KUKA KRL program: EPS_2_25748_MH05A_A_20260121065902.src

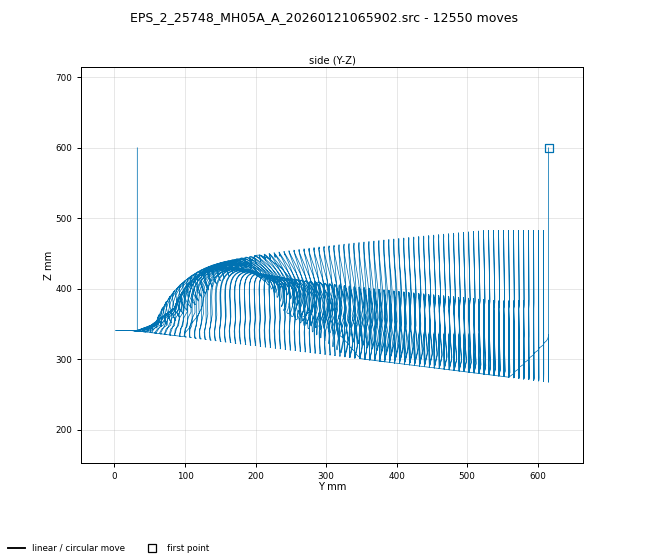
[picture p0: tool path of EPS_2_25748_MH05A_A_20260121065902.src, 12550 of 12552 moves have a stored position in this frame; points joined in program order, loops and branches not executed]
&ACCESS RVP
&REL 4
&COMMENT QRS 19112012
&PARAM EDITMASK = *
DEF PART()
EXT BAS (BAS_COMMAND :IN,REAL :IN )
INT I
BAS (#INITMOV,0 )

;KUKA QRS Post kuka4.cps  Date:22-06-2017 !

File_ID=3004

QRS_PRE_INIT()

;Init var - Until changes are made in qrs_pre_init
Outlet_Square_prg=0
Inlet_1_Square_prg=0
Inlet_2_Square_prg=0
Inlet_3_Square_prg=0
Inlet_4_Square_prg=0
Inlet_5_Square_prg=0

Outlet_1={X 0.000, Y 526.370, Z 382.500, B 0.000, E1 0.000 }
Inlet_1={X 0.000, Y 541.370, Z 332.500, B 0.000, E1 90.000 }
Inlet_2={X 0.000, Y 541.370, Z 332.500, B 0.000, E1 270.000 }
Outlet_1_type=201
Inlet_1_type=101
Inlet_2_type=101
;QRS#1=Sidecore dimensions
;QRS#2=200-8" PVC SDR 35
;QRS#3=100-4" PVC SDR 28
;QRS#4=100-4" PVC SDR 28
;QRS#5=
;QRS#6=
;QRS#7=
;QRS#8=
;QRS#9=12-08 PSX
;QRS#10=8QRS PSX
;QRS#11=8QRS PSX
;QRS#12=
;QRS#13=
;QRS#14=
;QRS#15=
;QRS#16=1220x127x762 2,5'
;QRS#17=EPS Height
;QRS#18=483
;QRS#19=*
;QRS#20= UPDATED VERSION 22-06-2017
;QRS#21=*
Outlet_Square=0100
Inlet_1_Square=045
Inlet_2_Square=045
Inlet_3_Square=0
Inlet_4_Square=0
Inlet_5_Square=0
Mill_Square=1
Outlet_Square_Prg=204
Inlet_1_Square_prg=201
Inlet_2_Square_prg=201

QRS_INIT()

$ADVANCE=5

; T1
PTP {E1 173.437,E2 173.437}
PTP {X 0,Y 615.487,A -85,B 0,C 180,E1 173.437,E2 173.437,E3 0,E4 0,E5 0,E6 0}
QRS_SPEED_INIT()
LIN {X 0,Y 615.487,Z 600,A -85,B 0,C 180,E1 173.437,E2 173.437,E3 0,E4 0,E5 0,E6 0} C_VEL
LIN {X 0,Y 615.487,Z 356.487,A -85,B 0,C 180,E1 173.437,E2 173.437} C_VEL
LIN {X 0,Y 615.487,Z 335.835,A -85,B 0,C 180,E1 173.437,E2 173.437} C_VEL
LIN {X 0,Y 615.487,Z 335.142,A -85,B 0,C 180,E1 173.425,E2 173.425} C_VEL
LIN {X 0,Y 615.489,Z 327.199,A -85,B 0,C 180,E1 173.165,E2 173.165} C_VEL
LIN {X 0,Y 615.468,Z 320.809,A -85,B 0,C 180,E1 170.802,E2 170.802} C_VEL
LIN {X 0,Y 615.487,Z 313.625,A -85,B 0,C 180,E1 168.14,E2 168.14} C_VEL
LIN {X 0,Y 615.472,Z 306.465,A -85,B 0,C 180,E1 165.452,E2 165.452} C_VEL
LIN {X 0,Y 615.459,Z 301.091,A -85,B 0,C 180,E1 163.414,E2 163.414} C_VEL
LIN {X 0,Y 615.449,Z 295.711,A -85,B 0,C 180,E1 161.354,E2 161.354} C_VEL
LIN {X 0,Y 615.488,Z 288.516,A -85,B 0,C 180,E1 158.569,E2 158.569} C_VEL
LIN {X 0,Y 615.439,Z 281.35,A -85,B 0,C 180,E1 155.727,E2 155.727} C_VEL
LIN {X 0,Y 615.424,Z 275.957,A -85,B 0,C 180,E1 153.554,E2 153.554} C_VEL
LIN {X 0,Y 615.496,Z 270.47,A -85,B 0,C 180,E1 151.344,E2 151.344} C_VEL
LIN {X 0,Y 615.454,Z 267.7,A -85,B 0,C 180,E1 150.211,E2 150.211} C_VEL
LIN {X 0,Y 615.419,Z 267.7,A -85,B 0,C 180,E1 147.54,E2 147.54} C_VEL
LIN {X 0,Y 615.453,Z 267.7,A -85,B 0,C 180,E1 145.184,E2 145.184} C_VEL
LIN {X 0,Y 615.487,Z 267.696,A -85,B 0,C 180,E1 142.759,E2 142.759} C_VEL
LIN {X 0,Y 615.437,Z 267.696,A -85,B 0,C 180,E1 140.248,E2 140.248} C_VEL
LIN {X 0,Y 615.459,Z 267.698,A -85,B 0,C 180,E1 137.646,E2 137.646} C_VEL
LIN {X 0,Y 615.492,Z 267.688,A -85,B 0,C 180,E1 134.934,E2 134.934} C_VEL
LIN {X 0,Y 615.453,Z 267.693,A -85,B 0,C 180,E1 132.356,E2 132.356} C_VEL
LIN {X 0,Y 615.497,Z 267.7,A -85,B 0,C 180,E1 129.75,E2 129.75} C_VEL
LIN {X 0,Y 615.478,Z 267.686,A -85,B 0,C 180,E1 126.938,E2 126.938} C_VEL
LIN {X 0,Y 615.495,Z 267.7,A -85,B 0,C 180,E1 124.022,E2 124.022} C_VEL
LIN {X 0,Y 615.484,Z 267.685,A -85,B 0,C 180,E1 121.088,E2 121.088} C_VEL
LIN {X 0,Y 615.494,Z 267.699,A -85,B 0,C 180,E1 118.454,E2 118.454} C_VEL
LIN {X 0,Y 615.485,Z 267.685,A -85,B 0,C 180,E1 115.571,E2 115.571} C_VEL
LIN {X 0,Y 615.492,Z 267.697,A -85,B 0,C 180,E1 112.844,E2 112.844} C_VEL
LIN {X 0,Y 615.476,Z 267.697,A -85,B 0,C 180,E1 110.558,E2 110.558} C_VEL
LIN {X 0,Y 615.468,Z 267.688,A -85,B 0,C 180,E1 107.958,E2 107.958} C_VEL
LIN {X 0,Y 615.497,Z 267.698,A -85,B 0,C 180,E1 105.226,E2 105.226} C_VEL
LIN {X 0,Y 615.447,Z 267.694,A -85,B 0,C 180,E1 102.531,E2 102.531} C_VEL
LIN {X 0,Y 615.489,Z 267.69,A -85,B 0,C 180,E1 99.862,E2 99.862} C_VEL
LIN {X 0,Y 615.455,Z 267.699,A -85,B 0,C 180,E1 97.216,E2 97.216} C_VEL
LIN {X 0,Y 615.445,Z 267.699,A -85,B 0,C 180,E1 95.242,E2 95.242} C_VEL
LIN {X 0,Y 615.436,Z 267.699,A -85,B 0,C 180,E1 93.273,E2 93.273} C_VEL
LIN {X 0,Y 615.428,Z 267.7,A -85,B 0,C 180,E1 91.309,E2 91.309} C_VEL
LIN {X 0,Y 615.426,Z 267.7,A -85,B 0,C 180,E1 89.346,E2 89.346} C_VEL
LIN {X 0,Y 615.429,Z 267.698,A -85,B 0,C 180,E1 87.382,E2 87.382} C_VEL
LIN {X 0,Y 615.433,Z 267.697,A -85,B 0,C 180,E1 85.415,E2 85.415} C_VEL
LIN {X 0,Y 615.436,Z 267.696,A -85,B 0,C 180,E1 83.443,E2 83.443} C_VEL
LIN {X 0,Y 615.465,Z 267.7,A -85,B 0,C 180,E1 80.801,E2 80.801} C_VEL
LIN {X 0,Y 615.481,Z 267.689,A -85,B 0,C 180,E1 78.139,E2 78.139} C_VEL
LIN {X 0,Y 615.455,Z 267.694,A -85,B 0,C 180,E1 75.45,E2 75.45} C_VEL
LIN {X 0,Y 615.489,Z 267.694,A -85,B 0,C 180,E1 72.729,E2 72.729} C_VEL
LIN {X 0,Y 615.467,Z 267.689,A -85,B 0,C 180,E1 69.966,E2 69.966} C_VEL
LIN {X 0,Y 615.474,Z 267.695,A -85,B 0,C 180,E1 67.653,E2 67.653} C_VEL
LIN {X 0,Y 615.483,Z 267.691,A -85,B 0,C 180,E1 65.008,E2 65.008} C_VEL
LIN {X 0,Y 615.484,Z 267.686,A -85,B 0,C 180,E1 62.823,E2 62.823} C_VEL
LIN {X 0,Y 615.481,Z 267.691,A -85,B 0,C 180,E1 60.204,E2 60.204} C_VEL
LIN {X 0,Y 615.476,Z 267.695,A -85,B 0,C 180,E1 57.542,E2 57.542} C_VEL
LIN {X 0,Y 615.471,Z 267.688,A -85,B 0,C 180,E1 55.184,E2 55.184} C_VEL
LIN {X 0,Y 615.495,Z 267.685,A -85,B 0,C 180,E1 52.758,E2 52.758} C_VEL
LIN {X 0,Y 615.464,Z 267.696,A -85,B 0,C 180,E1 49.912,E2 49.912} C_VEL
LIN {X 0,Y 615.451,Z 267.693,A -85,B 0,C 180,E1 47.644,E2 47.644} C_VEL
LIN {X 0,Y 615.493,Z 267.691,A -85,B 0,C 180,E1 44.932,E2 44.932} C_VEL
LIN {X 0,Y 615.456,Z 267.698,A -85,B 0,C 180,E1 42.354,E2 42.354} C_VEL
LIN {X 0,Y 615.435,Z 267.696,A -85,B 0,C 180,E1 39.753,E2 39.753} C_VEL
LIN {X 0,Y 615.487,Z 267.696,A -85,B 0,C 180,E1 37.241,E2 37.241} C_VEL
LIN {X 0,Y 615.437,Z 267.7,A -85,B 0,C 180,E1 34.693,E2 34.693} C_VEL
LIN {X 0,Y 615.418,Z 267.7,A -85,B 0,C 180,E1 32.32,E2 32.32} C_VEL
LIN {X 0,Y 615.467,Z 267.832,A -85,B 0,C 180,E1 29.693,E2 29.693} C_VEL
LIN {X 0,Y 615.464,Z 273.932,A -85,B 0,C 180,E1 27.177,E2 27.177} C_VEL
LIN {X 0,Y 615.444,Z 279.32,A -85,B 0,C 180,E1 24.992,E2 24.992} C_VEL
LIN {X 0,Y 615.435,Z 284.707,A -85,B 0,C 180,E1 22.845,E2 22.845} C_VEL
LIN {X 0,Y 615.435,Z 290.579,A -85,B 0,C 180,E1 20.543,E2 20.543} C_VEL
LIN {X 0,Y 615.494,Z 297.255,A -85,B 0,C 180,E1 17.956,E2 17.956} C_VEL
LIN {X 0,Y 615.458,Z 304.432,A -85,B 0,C 180,E1 15.226,E2 15.226} C_VEL
LIN {X 0,Y 615.458,Z 309.811,A -85,B 0,C 180,E1 13.201,E2 13.201} C_VEL
LIN {X 0,Y 615.486,Z 316.97,A -85,B 0,C 180,E1 10.526,E2 10.526} C_VEL
LIN {X 0,Y 615.488,Z 324.129,A -85,B 0,C 180,E1 7.875,E2 7.875} C_VEL
LIN {X 0,Y 615.484,Z 327.224,A -85,B 0,C 180,E1 6.736,E2 6.736} C_VEL
LIN {X 0,Y 615.489,Z 337.548,A -85,B 0,C 180,E1 6.391,E2 6.391} C_VEL
LIN {X 0,Y 615.493,Z 345.958,A -85,B 0,C 180,E1 5.98,E2 5.98} C_VEL
LIN {X 0,Y 615.473,Z 353.687,A -85,B 0,C 180,E1 5.487,E2 5.487} C_VEL
LIN {X 0,Y 615.479,Z 360.528,A -85,B 0,C 180,E1 4.912,E2 4.912} C_VEL
LIN {X 0,Y 615.497,Z 366.675,A -85,B 0,C 180,E1 4.255,E2 4.255} C_VEL
LIN {X 0,Y 615.497,Z 371.521,A -85,B 0,C 180,E1 3.6,E2 3.6} C_VEL
LIN {X 0,Y 615.496,Z 375.254,A -85,B 0,C 180,E1 2.944,E2 2.944} C_VEL
LIN {X 0,Y 615.5,Z 379.232,A -85,B 0,C 180,E1 1.962,E2 1.962} C_VEL
LIN {X 0,Y 615.495,Z 380.966,A -85,B 0,C 180,E1 1.308,E2 1.308} C_VEL
LIN {X 0,Y 615.496,Z 382.005,A -85,B 0,C 180,E1 0.653,E2 0.653} C_VEL
LIN {X 0,Y 615.495,Z 382.384,A -85,B 0,C 180,E1 -0.001,E2 -0.001} C_VEL
LIN {X 0,Y 615.496,Z 382.104,A -85,B 0,C 180,E1 -0.655,E2 -0.655} C_VEL
LIN {X 0,Y 615.497,Z 381.164,A -85,B 0,C 180,E1 -1.309,E2 -1.309} C_VEL
LIN {X 0,Y 615.5,Z 379.533,A -85,B 0,C 180,E1 -1.964,E2 -1.964} C_VEL
LIN {X 0,Y 615.498,Z 375.659,A -85,B 0,C 180,E1 -2.946,E2 -2.946} C_VEL
LIN {X 0,Y 615.5,Z 371.006,A -85,B 0,C 180,E1 -3.765,E2 -3.765} C_VEL
LIN {X 0,Y 615.498,Z 366.023,A -85,B 0,C 180,E1 -4.421,E2 -4.421} C_VEL
LIN {X 0,Y 615.481,Z 359.747,A -85,B 0,C 180,E1 -5.078,E2 -5.078} C_VEL
LIN {X 0,Y 615.481,Z 352.578,A -85,B 0,C 180,E1 -5.653,E2 -5.653} C_VEL
LIN {X 0,Y 615.485,Z 344.591,A -85,B 0,C 180,E1 -6.146,E2 -6.146} C_VEL
LIN {X 0,Y 615.487,Z 335.142,A -85,B 0,C 180,E1 -6.575,E2 -6.575} C_VEL
LIN {X 0,Y 615.489,Z 327.197,A -85,B 0,C 180,E1 -6.835,E2 -6.835} C_VEL
LIN {X 0,Y 615.468,Z 320.805,A -85,B 0,C 180,E1 -9.2,E2 -9.2} C_VEL
LIN {X 0,Y 615.487,Z 313.62,A -85,B 0,C 180,E1 -11.862,E2 -11.862} C_VEL
LIN {X 0,Y 615.471,Z 306.46,A -85,B 0,C 180,E1 -14.55,E2 -14.55} C_VEL
LIN {X 0,Y 615.459,Z 301.086,A -85,B 0,C 180,E1 -16.588,E2 -16.588} C_VEL
LIN {X 0,Y 615.449,Z 295.706,A -85,B 0,C 180,E1 -18.648,E2 -18.648} C_VEL
LIN {X 0,Y 615.488,Z 288.511,A -85,B 0,C 180,E1 -21.433,E2 -21.433} C_VEL
LIN {X 0,Y 615.439,Z 281.345,A -85,B 0,C 180,E1 -24.275,E2 -24.275} C_VEL
LIN {X 0,Y 615.424,Z 275.952,A -85,B 0,C 180,E1 -26.448,E2 -26.448} C_VEL
LIN {X 0,Y 615.494,Z 270.525,A -85,B 0,C 180,E1 -28.658,E2 -28.658} C_VEL
LIN {X 0,Y 615.474,Z 267.701,A -85,B 0,C 180,E1 -29.838,E2 -29.838} C_VEL
LIN {X 0,Y 615.483,Z 267.7,A -85,B 0,C 180,E1 -32.458,E2 -32.458} C_VEL
LIN {X 0,Y 615.499,Z 267.7,A -85,B 0,C 180,E1 -34.815,E2 -34.815} C_VEL
LIN {X 0,Y 615.494,Z 267.696,A -85,B 0,C 180,E1 -37.242,E2 -37.242} C_VEL
LIN {X 0,Y 615.497,Z 267.7,A -85,B 0,C 180,E1 -40.09,E2 -40.09} C_VEL
LIN {X 0,Y 615.492,Z 267.699,A -85,B 0,C 180,E1 -43.048,E2 -43.048} C_VEL
LIN {X 0,Y 615.474,Z 267.7,A -85,B 0,C 180,E1 -45.849,E2 -45.849} C_VEL
LIN {X 0,Y 615.495,Z 267.7,A -85,B 0,C 180,E1 -48.527,E2 -48.527} C_VEL
LIN {X 0,Y 615.489,Z 267.697,A -85,B 0,C 180,E1 -51.096,E2 -51.096} C_VEL
LIN {X 0,Y 615.49,Z 267.7,A -85,B 0,C 180,E1 -53.575,E2 -53.575} C_VEL
LIN {X 0,Y 615.484,Z 267.698,A -85,B 0,C 180,E1 -56.467,E2 -56.467} C_VEL
LIN {X 0,Y 615.487,Z 267.701,A -85,B 0,C 180,E1 -59.08,E2 -59.08} C_VEL
LIN {X 0,Y 615.475,Z 267.7,A -85,B 0,C 180,E1 -61.553,E2 -61.553} C_VEL
LIN {X 0,Y 615.499,Z 267.84,A -85,B 0,C 180,E1 -62.593,E2 -62.593} C_VEL
LIN {X 0,Y 615.489,Z 285.437,A -85,B 0,C 180,E1 -65.369,E2 -65.369} C_VEL
LIN {X 0,Y 615.479,Z 303.892,A -85,B 0,C 180,E1 -68.216,E2 -68.216} C_VEL
LIN {X 0,Y 615.48,Z 322.328,A -85,B 0,C 180,E1 -71.008,E2 -71.008} C_VEL
LIN {X 0,Y 615.475,Z 339.53,A -85,B 0,C 180,E1 -73.574,E2 -73.574} C_VEL
LIN {X 0,Y 615.493,Z 357.991,A -85,B 0,C 180,E1 -76.294,E2 -76.294} C_VEL
LIN {X 0,Y 615.497,Z 371.777,A -85,B 0,C 180,E1 -78.306,E2 -78.306} C_VEL
LIN {X 0,Y 615.48,Z 386.239,A -85,B 0,C 180,E1 -78.557,E2 -78.557} C_VEL
LIN {X 0,Y 615.474,Z 399.368,A -85,B 0,C 180,E1 -78.923,E2 -78.923} C_VEL
LIN {X 0,Y 615.487,Z 411.143,A -85,B 0,C 180,E1 -79.384,E2 -79.384} C_VEL
LIN {X 0,Y 615.486,Z 422.574,A -85,B 0,C 180,E1 -79.972,E2 -79.972} C_VEL
LIN {X 0,Y 615.499,Z 434.02,A -85,B 0,C 180,E1 -80.718,E2 -80.718} C_VEL
LIN {X 0,Y 615.498,Z 443.257,A -85,B 0,C 180,E1 -81.463,E2 -81.463} C_VEL
LIN {X 0,Y 615.5,Z 451.653,A -85,B 0,C 180,E1 -82.29,E2 -82.29} C_VEL
LIN {X 0,Y 615.497,Z 459.691,A -85,B 0,C 180,E1 -83.259,E2 -83.259} C_VEL
LIN {X 0,Y 615.499,Z 465.422,A -85,B 0,C 180,E1 -84.102,E2 -84.102} C_VEL
LIN {X 0,Y 615.496,Z 470.872,A -85,B 0,C 180,E1 -85.087,E2 -85.087} C_VEL
LIN {X 0,Y 615.497,Z 475.141,A -85,B 0,C 180,E1 -86.072,E2 -86.072} C_VEL
LIN {X 0,Y 615.494,Z 477.399,A -85,B 0,C 180,E1 -86.727,E2 -86.727} C_VEL
LIN {X 0,Y 615.497,Z 479.233,A -85,B 0,C 180,E1 -87.382,E2 -87.382} C_VEL
LIN {X 0,Y 615.5,Z 480.607,A -85,B 0,C 180,E1 -88.037,E2 -88.037} C_VEL
LIN {X 0,Y 615.496,Z 482.173,A -85,B 0,C 180,E1 -89.346,E2 -89.346} C_VEL
LIN {X 0,Y 615.494,Z 482.389,A -85,B 0,C 180,E1 -90,E2 -90} C_VEL
LIN {X 0,Y 615.495,Z 481.58,A -85,B 0,C 180,E1 -91.309,E2 -91.309} C_VEL
LIN {X 0,Y 615.5,Z 480.607,A -85,B 0,C 180,E1 -91.963,E2 -91.963} C_VEL
LIN {X 0,Y 615.497,Z 479.233,A -85,B 0,C 180,E1 -92.618,E2 -92.618} C_VEL
LIN {X 0,Y 615.496,Z 476.349,A -85,B 0,C 180,E1 -93.601,E2 -93.601} C_VEL
LIN {X 0,Y 615.498,Z 472.441,A -85,B 0,C 180,E1 -94.584,E2 -94.584} C_VEL
LIN {X 0,Y 615.499,Z 467.405,A -85,B 0,C 180,E1 -95.57,E2 -95.57} C_VEL
LIN {X 0,Y 615.497,Z 460.871,A -85,B 0,C 180,E1 -96.583,E2 -96.583} C_VEL
LIN {X 0,Y 615.497,Z 453.133,A -85,B 0,C 180,E1 -97.545,E2 -97.545} C_VEL
LIN {X 0,Y 615.498,Z 445.044,A -85,B 0,C 180,E1 -98.371,E2 -98.371} C_VEL
LIN {X 0,Y 615.499,Z 435.167,A -85,B 0,C 180,E1 -99.199,E2 -99.199} C_VEL
LIN {X 0,Y 615.49,Z 423.98,A -85,B 0,C 180,E1 -99.945,E2 -99.945} C_VEL
LIN {X 0,Y 615.487,Z 413.021,A -85,B 0,C 180,E1 -100.527,E2 -100.527} C_VEL
LIN {X 0,Y 615.475,Z 400.543,A -85,B 0,C 180,E1 -101.038,E2 -101.038} C_VEL
LIN {X 0,Y 615.478,Z 388.064,A -85,B 0,C 180,E1 -101.402,E2 -101.402} C_VEL
LIN {X 0,Y 615.495,Z 374.459,A -85,B 0,C 180,E1 -101.652,E2 -101.652} C_VEL
LIN {X 0,Y 615.497,Z 371.777,A -85,B 0,C 180,E1 -101.694,E2 -101.694} C_VEL
LIN {X 0,Y 615.474,Z 352.245,A -85,B 0,C 180,E1 -104.549,E2 -104.549} C_VEL
LIN {X 0,Y 615.494,Z 333.841,A -85,B 0,C 180,E1 -107.27,E2 -107.27} C_VEL
LIN {X 0,Y 615.486,Z 315.416,A -85,B 0,C 180,E1 -110.033,E2 -110.033} C_VEL
LIN {X 0,Y 615.492,Z 298.599,A -85,B 0,C 180,E1 -112.595,E2 -112.595} C_VEL
LIN {X 0,Y 615.496,Z 279.441,A -85,B 0,C 180,E1 -115.57,E2 -115.57} C_VEL
LIN {X 0,Y 615.498,Z 267.695,A -85,B 0,C 180,E1 -117.453,E2 -117.453} C_VEL
LIN {X 0,Y 615.487,Z 267.7,A -85,B 0,C 180,E1 -120.16,E2 -120.16} C_VEL
LIN {X 0,Y 615.477,Z 267.7,A -85,B 0,C 180,E1 -122.458,E2 -122.458} C_VEL
LIN {X 0,Y 615.479,Z 267.699,A -85,B 0,C 180,E1 -124.816,E2 -124.816} C_VEL
LIN {X 0,Y 615.498,Z 267.697,A -85,B 0,C 180,E1 -127.242,E2 -127.242} C_VEL
LIN {X 0,Y 615.474,Z 267.7,A -85,B 0,C 180,E1 -130.087,E2 -130.087} C_VEL
LIN {X 0,Y 615.473,Z 267.701,A -85,B 0,C 180,E1 -132.355,E2 -132.355} C_VEL
LIN {X 0,Y 615.491,Z 267.699,A -85,B 0,C 180,E1 -135.068,E2 -135.068} C_VEL
LIN {X 0,Y 615.483,Z 267.701,A -85,B 0,C 180,E1 -137.921,E2 -137.921} C_VEL
LIN {X 0,Y 615.494,Z 267.7,A -85,B 0,C 180,E1 -140.25,E2 -140.25} C_VEL
LIN {X 0,Y 615.493,Z 267.697,A -85,B 0,C 180,E1 -143.063,E2 -143.063} C_VEL
LIN {X 0,Y 615.487,Z 267.699,A -85,B 0,C 180,E1 -145.3,E2 -145.3} C_VEL
LIN {X 0,Y 615.494,Z 267.701,A -85,B 0,C 180,E1 -147.669,E2 -147.669} C_VEL
LIN {X 0,Y 615.491,Z 267.747,A -85,B 0,C 180,E1 -150.545,E2 -150.545} C_VEL
LIN {X 0,Y 615.49,Z 272.137,A -85,B 0,C 180,E1 -152.084,E2 -152.084} C_VEL
LIN {X 0,Y 615.444,Z 279.315,A -85,B 0,C 180,E1 -155.006,E2 -155.006} C_VEL
LIN {X 0,Y 615.435,Z 284.702,A -85,B 0,C 180,E1 -157.153,E2 -157.153} C_VEL
LIN {X 0,Y 615.435,Z 290.579,A -85,B 0,C 180,E1 -159.457,E2 -159.457} C_VEL
LIN {X 0,Y 615.494,Z 297.25,A -85,B 0,C 180,E1 -162.043,E2 -162.043} C_VEL
LIN {X 0,Y 615.458,Z 304.428,A -85,B 0,C 180,E1 -164.773,E2 -164.773} C_VEL
LIN {X 0,Y 615.458,Z 309.806,A -85,B 0,C 180,E1 -166.797,E2 -166.797} C_VEL
LIN {X 0,Y 615.486,Z 316.966,A -85,B 0,C 180,E1 -169.472,E2 -169.472} C_VEL
LIN {X 0,Y 615.488,Z 324.125,A -85,B 0,C 180,E1 -172.124,E2 -172.124} C_VEL
LIN {X 0,Y 615.484,Z 327.223,A -85,B 0,C 180,E1 -173.264,E2 -173.264} C_VEL
LIN {X 0,Y 615.489,Z 337.51,A -85,B 0,C 180,E1 -173.607,E2 -173.607} C_VEL
LIN {X 0,Y 615.493,Z 345.927,A -85,B 0,C 180,E1 -174.019,E2 -174.019} C_VEL
LIN {X 0,Y 615.473,Z 353.663,A -85,B 0,C 180,E1 -174.511,E2 -174.511} C_VEL
LIN {X 0,Y 615.479,Z 360.51,A -85,B 0,C 180,E1 -175.086,E2 -175.086} C_VEL
LIN {X 0,Y 615.497,Z 366.661,A -85,B 0,C 180,E1 -175.743,E2 -175.743} C_VEL
LIN {X 0,Y 615.497,Z 371.51,A -85,B 0,C 180,E1 -176.399,E2 -176.399} C_VEL
LIN {X 0,Y 615.496,Z 375.246,A -85,B 0,C 180,E1 -177.054,E2 -177.054} C_VEL
LIN {X 0,Y 615.5,Z 379.226,A -85,B 0,C 180,E1 -178.036,E2 -178.036} C_VEL
LIN {X 0,Y 615.495,Z 380.962,A -85,B 0,C 180,E1 -178.691,E2 -178.691} C_VEL
LIN {X 0,Y 615.496,Z 382.003,A -85,B 0,C 180,E1 -179.345,E2 -179.345} C_VEL
LIN {X 0,Y 615.495,Z 382.384,A -85,B 0,C 180,E1 -179.999,E2 -179.999} C_VEL
LIN {X 0,Y 615.496,Z 382.106,A -85,B 0,C 180,E1 -180.653,E2 -180.653} C_VEL
LIN {X 0,Y 615.497,Z 381.167,A -85,B 0,C 180,E1 -181.308,E2 -181.308} C_VEL
LIN {X 0,Y 615.5,Z 379.538,A -85,B 0,C 180,E1 -181.962,E2 -181.962} C_VEL
LIN {X 0,Y 615.497,Z 377.17,A -85,B 0,C 180,E1 -182.617,E2 -182.617} C_VEL
LIN {X 0,Y 615.498,Z 372.077,A -85,B 0,C 180,E1 -183.6,E2 -183.6} C_VEL
LIN {X 0,Y 615.499,Z 366.038,A -85,B 0,C 180,E1 -184.42,E2 -184.42} C_VEL
LIN {X 0,Y 615.482,Z 359.765,A -85,B 0,C 180,E1 -185.076,E2 -185.076} C_VEL
LIN {X 0,Y 615.481,Z 352.603,A -85,B 0,C 180,E1 -185.651,E2 -185.651} C_VEL
LIN {X 0,Y 615.485,Z 344.622,A -85,B 0,C 180,E1 -186.144,E2 -186.144} C_VEL
LIN {X 0,Y 615.487,Z 335.142,A -85,B 0,C 180,E1 -186.575,E2 -186.575} C_VEL
LIN {X 0,Y 615.134,Z 331.885,A -85,B 0,C 180,E1 -186.751,E2 -186.751} C_VEL
LIN {X 0,Y 614.287,Z 329.277,A -85,B 0,C 180,E1 -187,E2 -187} C_VEL
LIN {X 0,Y 612.54,Z 326.422,A -85,B 0,C 180,E1 -187.454,E2 -187.454} C_VEL
LIN {X 0,Y 610.632,Z 324.727,A -85,B 0,C 180,E1 -187.981,E2 -187.981} C_VEL
LIN {X 0,Y 608.713,Z 322.769,A -85,B 0,C 180,E1 -188.74,E2 -188.74} C_VEL
LIN {X 0,Y 608.404,Z 321.715,A -85,B 0,C 180,E1 -189.128,E2 -189.128} C_VEL
LIN {X 0,Y 608.405,Z 315.822,A -85,B 0,C 180,E1 -191.324,E2 -191.324} C_VEL
LIN {X 0,Y 608.43,Z 308.603,A -85,B 0,C 180,E1 -194.037,E2 -194.037} C_VEL
LIN {X 0,Y 608.397,Z 301.383,A -85,B 0,C 180,E1 -196.785,E2 -196.785} C_VEL
LIN {X 0,Y 608.443,Z 294.164,A -85,B 0,C 180,E1 -199.57,E2 -199.57} C_VEL
LIN {X 0,Y 608.393,Z 286.81,A -85,B 0,C 180,E1 -202.46,E2 -202.46} C_VEL
LIN {X 0,Y 608.417,Z 281.529,A -85,B 0,C 180,E1 -204.571,E2 -204.571} C_VEL
LIN {X 0,Y 608.46,Z 275.067,A -85,B 0,C 180,E1 -207.203,E2 -207.203} C_VEL
LIN {X 0,Y 608.439,Z 268.694,A -85,B 0,C 180,E1 -209.78,E2 -209.78} C_VEL
LIN {X 0,Y 608.405,Z 268.695,A -85,B 0,C 180,E1 -212.514,E2 -212.514} C_VEL
LIN {X 0,Y 608.418,Z 268.698,A -85,B 0,C 180,E1 -214.901,E2 -214.901} C_VEL
LIN {X 0,Y 608.431,Z 268.691,A -85,B 0,C 180,E1 -217.747,E2 -217.747} C_VEL
LIN {X 0,Y 608.426,Z 268.694,A -85,B 0,C 180,E1 -220.326,E2 -220.326} C_VEL
LIN {X 0,Y 608.462,Z 268.688,A -85,B 0,C 180,E1 -223.308,E2 -223.308} C_VEL
LIN {X 0,Y 608.447,Z 268.693,A -85,B 0,C 180,E1 -226.128,E2 -226.128} C_VEL
LIN {X 0,Y 608.459,Z 268.69,A -85,B 0,C 180,E1 -228.823,E2 -228.823} C_VEL
LIN {X 0,Y 608.459,Z 268.688,A -85,B 0,C 180,E1 -231.411,E2 -231.411} C_VEL
LIN {X 0,Y 608.471,Z 268.694,A -85,B 0,C 180,E1 -233.949,E2 -233.949} C_VEL
LIN {X 0,Y 608.466,Z 268.69,A -85,B 0,C 180,E1 -236.329,E2 -236.329} C_VEL
LIN {X 0,Y 608.47,Z 268.686,A -85,B 0,C 180,E1 -238.726,E2 -238.726} C_VEL
LIN {X 0,Y 608.473,Z 268.691,A -85,B 0,C 180,E1 -241.377,E2 -241.377} C_VEL
LIN {X 0,Y 608.443,Z 268.692,A -85,B 0,C 180,E1 -243.964,E2 -243.964} C_VEL
LIN {X 0,Y 608.452,Z 268.691,A -85,B 0,C 180,E1 -246.876,E2 -246.876} C_VEL
LIN {X 0,Y 608.46,Z 268.695,A -85,B 0,C 180,E1 -249.319,E2 -249.319} C_VEL
LIN {X 0,Y 608.432,Z 268.691,A -85,B 0,C 180,E1 -251.828,E2 -251.828} C_VEL
LIN {X 0,Y 608.474,Z 268.691,A -85,B 0,C 180,E1 -254.594,E2 -254.594} C_VEL
LIN {X 0,Y 608.448,Z 268.69,A -85,B 0,C 180,E1 -257.322,E2 -257.322} C_VEL
LIN {X 0,Y 608.45,Z 268.691,A -85,B 0,C 180,E1 -260.023,E2 -260.023} C_VEL
LIN {X 0,Y 608.426,Z 268.697,A -85,B 0,C 180,E1 -262.7,E2 -262.7} C_VEL
LIN {X 0,Y 608.431,Z 268.695,A -85,B 0,C 180,E1 -264.698,E2 -264.698} C_VEL
LIN {X 0,Y 608.423,Z 268.692,A -85,B 0,C 180,E1 -267.352,E2 -267.352} C_VEL
LIN {X 0,Y 608.465,Z 268.697,A -85,B 0,C 180,E1 -270,E2 -270} C_VEL
LIN {X 0,Y 608.424,Z 268.692,A -85,B 0,C 180,E1 -272.648,E2 -272.648} C_VEL
LIN {X 0,Y 608.433,Z 268.695,A -85,B 0,C 180,E1 -275.302,E2 -275.302} C_VEL
LIN {X 0,Y 608.468,Z 268.69,A -85,B 0,C 180,E1 -277.967,E2 -277.967} C_VEL
LIN {X 0,Y 608.427,Z 268.692,A -85,B 0,C 180,E1 -280.651,E2 -280.651} C_VEL
LIN {X 0,Y 608.469,Z 268.694,A -85,B 0,C 180,E1 -283.356,E2 -283.356} C_VEL
LIN {X 0,Y 608.443,Z 268.689,A -85,B 0,C 180,E1 -286.094,E2 -286.094} C_VEL
LIN {X 0,Y 608.448,Z 268.699,A -85,B 0,C 180,E1 -288.87,E2 -288.87} C_VEL
LIN {X 0,Y 608.466,Z 268.687,A -85,B 0,C 180,E1 -291.692,E2 -291.692} C_VEL
LIN {X 0,Y 608.446,Z 268.699,A -85,B 0,C 180,E1 -294.571,E2 -294.571} C_VEL
LIN {X 0,Y 608.475,Z 268.686,A -85,B 0,C 180,E1 -297.21,E2 -297.21} C_VEL
LIN {X 0,Y 608.465,Z 268.692,A -85,B 0,C 180,E1 -299.974,E2 -299.974} C_VEL
LIN {X 0,Y 608.452,Z 268.692,A -85,B 0,C 180,E1 -302.523,E2 -302.523} C_VEL
LIN {X 0,Y 608.464,Z 268.687,A -85,B 0,C 180,E1 -304.91,E2 -304.91} C_VEL
LIN {X 0,Y 608.465,Z 268.696,A -85,B 0,C 180,E1 -307.747,E2 -307.747} C_VEL
LIN {X 0,Y 608.428,Z 268.693,A -85,B 0,C 180,E1 -310.328,E2 -310.328} C_VEL
LIN {X 0,Y 608.45,Z 268.691,A -85,B 0,C 180,E1 -312.96,E2 -312.96} C_VEL
LIN {X 0,Y 608.428,Z 268.695,A -85,B 0,C 180,E1 -315.739,E2 -315.739} C_VEL
LIN {X 0,Y 608.423,Z 268.693,A -85,B 0,C 180,E1 -317.937,E2 -317.937} C_VEL
LIN {X 0,Y 608.439,Z 268.694,A -85,B 0,C 180,E1 -320.706,E2 -320.706} C_VEL
LIN {X 0,Y 608.449,Z 268.696,A -85,B 0,C 180,E1 -323.086,E2 -323.086} C_VEL
LIN {X 0,Y 608.42,Z 268.693,A -85,B 0,C 180,E1 -325.529,E2 -325.529} C_VEL
LIN {X 0,Y 608.416,Z 268.693,A -85,B 0,C 180,E1 -327.904,E2 -327.904} C_VEL
LIN {X 0,Y 608.458,Z 268.865,A -85,B 0,C 180,E1 -330.317,E2 -330.317} C_VEL
LIN {X 0,Y 608.457,Z 274.849,A -85,B 0,C 180,E1 -332.797,E2 -332.797} C_VEL
LIN {X 0,Y 608.411,Z 281.306,A -85,B 0,C 180,E1 -335.428,E2 -335.428} C_VEL
LIN {X 0,Y 608.431,Z 288.521,A -85,B 0,C 180,E1 -338.308,E2 -338.308} C_VEL
LIN {X 0,Y 608.409,Z 295.737,A -85,B 0,C 180,E1 -341.13,E2 -341.13} C_VEL
LIN {X 0,Y 608.44,Z 302.953,A -85,B 0,C 180,E1 -343.907,E2 -343.907} C_VEL
LIN {X 0,Y 608.411,Z 310.169,A -85,B 0,C 180,E1 -346.643,E2 -346.643} C_VEL
LIN {X 0,Y 608.419,Z 317.385,A -85,B 0,C 180,E1 -349.35,E2 -349.35} C_VEL
LIN {X 0,Y 608.419,Z 324.602,A -85,B 0,C 180,E1 -352.033,E2 -352.033} C_VEL
LIN {X 0,Y 608.446,Z 327.892,A -85,B 0,C 180,E1 -353.187,E2 -353.187} C_VEL
LIN {X 0,Y 608.477,Z 338.104,A -85,B 0,C 180,E1 -353.535,E2 -353.535} C_VEL
LIN {X 0,Y 608.464,Z 346.487,A -85,B 0,C 180,E1 -353.951,E2 -353.951} C_VEL
LIN {X 0,Y 608.438,Z 355.268,A -85,B 0,C 180,E1 -354.533,E2 -354.533} C_VEL
LIN {X 0,Y 608.456,Z 362.738,A -85,B 0,C 180,E1 -355.197,E2 -355.197} C_VEL
LIN {X 0,Y 608.437,Z 368.565,A -85,B 0,C 180,E1 -355.861,E2 -355.861} C_VEL
LIN {X 0,Y 608.451,Z 372.073,A -85,B 0,C 180,E1 -356.359,E2 -356.359} C_VEL
LIN {X 0,Y 608.451,Z 375.824,A -85,B 0,C 180,E1 -357.021,E2 -357.021} C_VEL
LIN {X 0,Y 608.445,Z 379.829,A -85,B 0,C 180,E1 -358.015,E2 -358.015} C_VEL
LIN {X 0,Y 608.448,Z 381.57,A -85,B 0,C 180,E1 -358.677,E2 -358.677} C_VEL
LIN {X 0,Y 608.439,Z 382.615,A -85,B 0,C 180,E1 -359.339,E2 -359.339} C_VEL
LIN {X 0,Y 608.435,Z 382.995,A -85,B 0,C 180,E1 -360.001,E2 -360.001} C_VEL
LIN {X 0,Y 608.438,Z 382.713,A -85,B 0,C 180,E1 -360.663,E2 -360.663} C_VEL
LIN {X 0,Y 608.449,Z 381.766,A -85,B 0,C 180,E1 -361.325,E2 -361.325} C_VEL
LIN {X 0,Y 608.445,Z 380.126,A -85,B 0,C 180,E1 -361.987,E2 -361.987} C_VEL
LIN {X 0,Y 608.429,Z 377.742,A -85,B 0,C 180,E1 -362.649,E2 -362.649} C_VEL
LIN {X 0,Y 608.452,Z 372.614,A -85,B 0,C 180,E1 -363.643,E2 -363.643} C_VEL
LIN {X 0,Y 608.451,Z 366.548,A -85,B 0,C 180,E1 -364.473,E2 -364.473} C_VEL
LIN {X 0,Y 608.429,Z 360.244,A -85,B 0,C 180,E1 -365.137,E2 -365.137} C_VEL
LIN {X 0,Y 608.463,Z 353.082,A -85,B 0,C 180,E1 -365.718,E2 -365.718} C_VEL
LIN {X 0,Y 608.445,Z 345.091,A -85,B 0,C 180,E1 -366.217,E2 -366.217} C_VEL
LIN {X 0,Y 608.466,Z 336.237,A -85,B 0,C 180,E1 -366.633,E2 -366.633} C_VEL
LIN {X 0,Y 608.428,Z 327.701,A -85,B 0,C 180,E1 -366.91,E2 -366.91} C_VEL
LIN {X 0,Y 608.402,Z 321.231,A -85,B 0,C 180,E1 -369.308,E2 -369.308} C_VEL
LIN {X 0,Y 608.432,Z 314.012,A -85,B 0,C 180,E1 -372.001,E2 -372.001} C_VEL
LIN {X 0,Y 608.429,Z 306.793,A -85,B 0,C 180,E1 -374.722,E2 -374.722} C_VEL
LIN {X 0,Y 608.423,Z 299.574,A -85,B 0,C 180,E1 -377.478,E2 -377.478} C_VEL
LIN {X 0,Y 608.422,Z 292.354,A -85,B 0,C 180,E1 -380.276,E2 -380.276} C_VEL
LIN {X 0,Y 608.427,Z 285.134,A -85,B 0,C 180,E1 -383.126,E2 -383.126} C_VEL
LIN {X 0,Y 608.419,Z 277.914,A -85,B 0,C 180,E1 -386.037,E2 -386.037} C_VEL
LIN {X 0,Y 608.482,Z 271.589,A -85,B 0,C 180,E1 -388.621,E2 -388.621} C_VEL
LIN {X 0,Y 608.455,Z 268.696,A -85,B 0,C 180,E1 -389.841,E2 -389.841} C_VEL
LIN {X 0,Y 608.46,Z 268.696,A -85,B 0,C 180,E1 -392.522,E2 -392.522} C_VEL
LIN {X 0,Y 608.45,Z 268.696,A -85,B 0,C 180,E1 -395.278,E2 -395.278} C_VEL
LIN {X 0,Y 608.472,Z 268.694,A -85,B 0,C 180,E1 -397.747,E2 -397.747} C_VEL
LIN {X 0,Y 608.451,Z 268.696,A -85,B 0,C 180,E1 -400.329,E2 -400.329} C_VEL
LIN {X 0,Y 608.457,Z 268.696,A -85,B 0,C 180,E1 -402.96,E2 -402.96} C_VEL
LIN {X 0,Y 608.448,Z 268.696,A -85,B 0,C 180,E1 -405.738,E2 -405.738} C_VEL
LIN {X 0,Y 608.47,Z 268.694,A -85,B 0,C 180,E1 -408.658,E2 -408.658} C_VEL
LIN {X 0,Y 608.464,Z 268.696,A -85,B 0,C 180,E1 -411.761,E2 -411.761} C_VEL
LIN {X 0,Y 608.447,Z 268.697,A -85,B 0,C 180,E1 -413.955,E2 -413.955} C_VEL
LIN {X 0,Y 608.452,Z 268.695,A -85,B 0,C 180,E1 -416.328,E2 -416.328} C_VEL
LIN {X 0,Y 608.452,Z 268.696,A -85,B 0,C 180,E1 -418.732,E2 -418.732} C_VEL
LIN {X 0,Y 608.467,Z 268.694,A -85,B 0,C 180,E1 -421.382,E2 -421.382} C_VEL
LIN {X 0,Y 608.481,Z 268.705,A -85,B 0,C 180,E1 -422.39,E2 -422.39} C_VEL
LIN {X 0,Y 608.603,Z 280.287,A -85,B 0,C 180,E1 -424.254,E2 -424.254} C_VEL
LIN {X 0,Y 608.557,Z 298.245,A -85,B 0,C 180,E1 -427.078,E2 -427.078} C_VEL
LIN {X 0,Y 608.533,Z 316.593,A -85,B 0,C 180,E1 -429.904,E2 -429.904} C_VEL
LIN {X 0,Y 608.507,Z 335.055,A -85,B 0,C 180,E1 -432.698,E2 -432.698} C_VEL
LIN {X 0,Y 608.463,Z 353.518,A -85,B 0,C 180,E1 -435.45,E2 -435.45} C_VEL
LIN {X 0,Y 608.482,Z 371.981,A -85,B 0,C 180,E1 -438.17,E2 -438.17} C_VEL
LIN {X 0,Y 608.544,Z 387.264,A -85,B 0,C 180,E1 -438.445,E2 -438.445} C_VEL
LIN {X 0,Y 608.519,Z 399.925,A -85,B 0,C 180,E1 -438.809,E2 -438.809} C_VEL
LIN {X 0,Y 608.51,Z 411.635,A -85,B 0,C 180,E1 -439.277,E2 -439.277} C_VEL
LIN {X 0,Y 608.494,Z 422.755,A -85,B 0,C 180,E1 -439.855,E2 -439.855} C_VEL
LIN {X 0,Y 608.504,Z 434.251,A -85,B 0,C 180,E1 -440.611,E2 -440.611} C_VEL
LIN {X 0,Y 608.472,Z 443.536,A -85,B 0,C 180,E1 -441.364,E2 -441.364} C_VEL
LIN {X 0,Y 608.456,Z 451.989,A -85,B 0,C 180,E1 -442.2,E2 -442.2} C_VEL
LIN {X 0,Y 608.462,Z 460.235,A -85,B 0,C 180,E1 -443.201,E2 -443.201} C_VEL
LIN {X 0,Y 608.438,Z 466.876,A -85,B 0,C 180,E1 -444.199,E2 -444.199} C_VEL
LIN {X 0,Y 608.432,Z 472.95,A -85,B 0,C 180,E1 -445.362,E2 -445.362} C_VEL
LIN {X 0,Y 608.449,Z 476.896,A -85,B 0,C 180,E1 -446.358,E2 -446.358} C_VEL
LIN {X 0,Y 608.425,Z 479.809,A -85,B 0,C 180,E1 -447.352,E2 -447.352} C_VEL
LIN {X 0,Y 608.445,Z 481.201,A -85,B 0,C 180,E1 -448.014,E2 -448.014} C_VEL
LIN {X 0,Y 608.438,Z 482.783,A -85,B 0,C 180,E1 -449.338,E2 -449.338} C_VEL
LIN {X 0,Y 608.434,Z 483,A -85,B 0,C 180,E1 -450,E2 -450} C_VEL
LIN {X 0,Y 608.448,Z 482.184,A -85,B 0,C 180,E1 -451.324,E2 -451.324} C_VEL
LIN {X 0,Y 608.445,Z 481.201,A -85,B 0,C 180,E1 -451.986,E2 -451.986} C_VEL
LIN {X 0,Y 608.425,Z 479.809,A -85,B 0,C 180,E1 -452.648,E2 -452.648} C_VEL
LIN {X 0,Y 608.449,Z 476.896,A -85,B 0,C 180,E1 -453.642,E2 -453.642} C_VEL
LIN {X 0,Y 608.432,Z 472.95,A -85,B 0,C 180,E1 -454.638,E2 -454.638} C_VEL
LIN {X 0,Y 608.438,Z 466.876,A -85,B 0,C 180,E1 -455.801,E2 -455.801} C_VEL
LIN {X 0,Y 608.462,Z 460.235,A -85,B 0,C 180,E1 -456.799,E2 -456.799} C_VEL
LIN {X 0,Y 608.456,Z 451.989,A -85,B 0,C 180,E1 -457.8,E2 -457.8} C_VEL
LIN {X 0,Y 608.472,Z 443.536,A -85,B 0,C 180,E1 -458.636,E2 -458.636} C_VEL
LIN {X 0,Y 608.481,Z 433.09,A -85,B 0,C 180,E1 -459.473,E2 -459.473} C_VEL
LIN {X 0,Y 608.494,Z 422.754,A -85,B 0,C 180,E1 -460.145,E2 -460.145} C_VEL
LIN {X 0,Y 608.51,Z 411.635,A -85,B 0,C 180,E1 -460.723,E2 -460.723} C_VEL
LIN {X 0,Y 608.519,Z 399.926,A -85,B 0,C 180,E1 -461.191,E2 -461.191} C_VEL
LIN {X 0,Y 608.544,Z 387.265,A -85,B 0,C 180,E1 -461.555,E2 -461.555} C_VEL
LIN {X 0,Y 608.57,Z 374.597,A -85,B 0,C 180,E1 -461.786,E2 -461.786} C_VEL
LIN {X 0,Y 608.484,Z 371.981,A -85,B 0,C 180,E1 -461.83,E2 -461.83} C_VEL
LIN {X 0,Y 608.479,Z 352.364,A -85,B 0,C 180,E1 -464.72,E2 -464.72} C_VEL
LIN {X 0,Y 608.51,Z 333.901,A -85,B 0,C 180,E1 -467.475,E2 -467.475} C_VEL
LIN {X 0,Y 608.517,Z 315.439,A -85,B 0,C 180,E1 -470.272,E2 -470.272} C_VEL
LIN {X 0,Y 608.57,Z 298.131,A -85,B 0,C 180,E1 -472.939,E2 -472.939} C_VEL
LIN {X 0,Y 608.613,Z 280.271,A -85,B 0,C 180,E1 -475.748,E2 -475.748} C_VEL
LIN {X 0,Y 608.481,Z 268.705,A -85,B 0,C 180,E1 -477.61,E2 -477.61} C_VEL
LIN {X 0,Y 608.471,Z 268.693,A -85,B 0,C 180,E1 -480.545,E2 -480.545} C_VEL
LIN {X 0,Y 608.456,Z 268.695,A -85,B 0,C 180,E1 -482.88,E2 -482.88} C_VEL
LIN {X 0,Y 608.437,Z 268.7,A -85,B 0,C 180,E1 -485.278,E2 -485.278} C_VEL
LIN {X 0,Y 608.464,Z 268.694,A -85,B 0,C 180,E1 -487.747,E2 -487.747} C_VEL
LIN {X 0,Y 608.445,Z 268.697,A -85,B 0,C 180,E1 -490.328,E2 -490.328} C_VEL
LIN {X 0,Y 608.477,Z 268.692,A -85,B 0,C 180,E1 -493.309,E2 -493.309} C_VEL
LIN {X 0,Y 608.473,Z 268.694,A -85,B 0,C 180,E1 -496.13,E2 -496.13} C_VEL
LIN {X 0,Y 608.456,Z 268.695,A -85,B 0,C 180,E1 -498.823,E2 -498.823} C_VEL
LIN {X 0,Y 608.44,Z 268.698,A -85,B 0,C 180,E1 -501.409,E2 -501.409} C_VEL
LIN {X 0,Y 608.448,Z 268.696,A -85,B 0,C 180,E1 -503.955,E2 -503.955} C_VEL
LIN {X 0,Y 608.449,Z 268.697,A -85,B 0,C 180,E1 -506.328,E2 -506.328} C_VEL
LIN {X 0,Y 608.449,Z 268.699,A -85,B 0,C 180,E1 -508.733,E2 -508.733} C_VEL
LIN {X 0,Y 608.439,Z 268.809,A -85,B 0,C 180,E1 -510.646,E2 -510.646} C_VEL
LIN {X 0,Y 608.438,Z 274.857,A -85,B 0,C 180,E1 -512.801,E2 -512.801} C_VEL
LIN {X 0,Y 608.383,Z 281.301,A -85,B 0,C 180,E1 -515.425,E2 -515.425} C_VEL
LIN {X 0,Y 608.388,Z 286.713,A -85,B 0,C 180,E1 -517.591,E2 -517.591} C_VEL
LIN {X 0,Y 608.439,Z 293.928,A -85,B 0,C 180,E1 -520.428,E2 -520.428} C_VEL
LIN {X 0,Y 608.421,Z 299.34,A -85,B 0,C 180,E1 -522.522,E2 -522.522} C_VEL
LIN {X 0,Y 608.403,Z 304.752,A -85,B 0,C 180,E1 -524.592,E2 -524.592} C_VEL
LIN {X 0,Y 608.411,Z 310.164,A -85,B 0,C 180,E1 -526.642,E2 -526.642} C_VEL
LIN {X 0,Y 608.419,Z 317.38,A -85,B 0,C 180,E1 -529.349,E2 -529.349} C_VEL
LIN {X 0,Y 608.42,Z 324.597,A -85,B 0,C 180,E1 -532.032,E2 -532.032} C_VEL
LIN {X 0,Y 608.43,Z 327.839,A -85,B 0,C 180,E1 -533.186,E2 -533.186} C_VEL
LIN {X 0,Y 608.479,Z 338.067,A -85,B 0,C 180,E1 -533.533,E2 -533.533} C_VEL
LIN {X 0,Y 608.464,Z 346.462,A -85,B 0,C 180,E1 -533.949,E2 -533.949} C_VEL
LIN {X 0,Y 608.438,Z 355.246,A -85,B 0,C 180,E1 -534.531,E2 -534.531} C_VEL
LIN {X 0,Y 608.456,Z 362.72,A -85,B 0,C 180,E1 -535.196,E2 -535.196} C_VEL
LIN {X 0,Y 608.437,Z 368.553,A -85,B 0,C 180,E1 -535.859,E2 -535.859} C_VEL
LIN {X 0,Y 608.451,Z 372.062,A -85,B 0,C 180,E1 -536.357,E2 -536.357} C_VEL
LIN {X 0,Y 608.451,Z 375.815,A -85,B 0,C 180,E1 -537.02,E2 -537.02} C_VEL
LIN {X 0,Y 608.445,Z 379.822,A -85,B 0,C 180,E1 -538.013,E2 -538.013} C_VEL
LIN {X 0,Y 608.448,Z 381.566,A -85,B 0,C 180,E1 -538.675,E2 -538.675} C_VEL
LIN {X 0,Y 608.439,Z 382.614,A -85,B 0,C 180,E1 -539.337,E2 -539.337} C_VEL
LIN {X 0,Y 608.435,Z 382.995,A -85,B 0,C 180,E1 -539.999,E2 -539.999} C_VEL
LIN {X 0,Y 608.438,Z 382.715,A -85,B 0,C 180,E1 -540.661,E2 -540.661} C_VEL
LIN {X 0,Y 608.449,Z 381.77,A -85,B 0,C 180,E1 -541.323,E2 -541.323} C_VEL
LIN {X 0,Y 608.445,Z 380.131,A -85,B 0,C 180,E1 -541.985,E2 -541.985} C_VEL
LIN {X 0,Y 608.429,Z 377.749,A -85,B 0,C 180,E1 -542.647,E2 -542.647} C_VEL
LIN {X 0,Y 608.452,Z 372.624,A -85,B 0,C 180,E1 -543.641,E2 -543.641} C_VEL
LIN {X 0,Y 608.452,Z 366.565,A -85,B 0,C 180,E1 -544.471,E2 -544.471} C_VEL
LIN {X 0,Y 608.429,Z 360.261,A -85,B 0,C 180,E1 -545.135,E2 -545.135} C_VEL
LIN {X 0,Y 608.462,Z 353.11,A -85,B 0,C 180,E1 -545.717,E2 -545.717} C_VEL
LIN {X 0,Y 608.445,Z 345.128,A -85,B 0,C 180,E1 -546.216,E2 -546.216} C_VEL
LIN {X 0,Y 608.477,Z 335.531,A -85,B 0,C 180,E1 -546.658,E2 -546.658} C_VEL
LIN {X 0,Y 608.428,Z 327.703,A -85,B 0,C 180,E1 -546.91,E2 -546.91} C_VEL
LIN {X 0,Y 608.404,Z 321.715,A -85,B 0,C 180,E1 -549.128,E2 -549.128} C_VEL
LIN {X 0,Y 607.724,Z 320.3,A -85,B 0,C 180,E1 -549.665,E2 -549.665} C_VEL
LIN {X 0,Y 604.832,Z 318.095,A -85,B 0,C 180,E1 -550.537,E2 -550.537} C_VEL
LIN {X 0,Y 602.411,Z 316.347,A -85,B 0,C 180,E1 -551.239,E2 -551.239} C_VEL
LIN {X 0,Y 601.397,Z 314.968,A -85,B 0,C 180,E1 -551.781,E2 -551.781} C_VEL
LIN {X 0,Y 601.329,Z 314.489,A -85,B 0,C 180,E1 -551.964,E2 -551.964} C_VEL
LIN {X 0,Y 601.348,Z 306.796,A -85,B 0,C 180,E1 -554.898,E2 -554.898} C_VEL
LIN {X 0,Y 601.353,Z 299.577,A -85,B 0,C 180,E1 -557.689,E2 -557.689} C_VEL
LIN {X 0,Y 601.366,Z 294.162,A -85,B 0,C 180,E1 -559.81,E2 -559.81} C_VEL
LIN {X 0,Y 601.351,Z 286.943,A -85,B 0,C 180,E1 -562.684,E2 -562.684} C_VEL
LIN {X 0,Y 601.412,Z 279.722,A -85,B 0,C 180,E1 -565.617,E2 -565.617} C_VEL
LIN {X 0,Y 601.376,Z 274.159,A -85,B 0,C 180,E1 -567.868,E2 -567.868} C_VEL
LIN {X 0,Y 601.396,Z 269.573,A -85,B 0,C 180,E1 -569.682,E2 -569.682} C_VEL
LIN {X 0,Y 601.379,Z 269.57,A -85,B 0,C 180,E1 -572.517,E2 -572.517} C_VEL
LIN {X 0,Y 601.368,Z 269.58,A -85,B 0,C 180,E1 -575.108,E2 -575.108} C_VEL
LIN {X 0,Y 601.425,Z 269.567,A -85,B 0,C 180,E1 -577.418,E2 -577.418} C_VEL
LIN {X 0,Y 601.372,Z 269.57,A -85,B 0,C 180,E1 -579.996,E2 -579.996} C_VEL
LIN {X 0,Y 601.401,Z 269.576,A -85,B 0,C 180,E1 -582.669,E2 -582.669} C_VEL
LIN {X 0,Y 601.39,Z 269.568,A -85,B 0,C 180,E1 -585.478,E2 -585.478} C_VEL
LIN {X 0,Y 601.419,Z 269.574,A -85,B 0,C 180,E1 -588.405,E2 -588.405} C_VEL
LIN {X 0,Y 601.435,Z 269.564,A -85,B 0,C 180,E1 -590.875,E2 -590.875} C_VEL
LIN {X 0,Y 601.435,Z 269.567,A -85,B 0,C 180,E1 -593.733,E2 -593.733} C_VEL
LIN {X 0,Y 601.426,Z 269.564,A -85,B 0,C 180,E1 -596.686,E2 -596.686} C_VEL
LIN {X 0,Y 601.425,Z 269.565,A -85,B 0,C 180,E1 -599.058,E2 -599.058} C_VEL
LIN {X 0,Y 601.432,Z 269.569,A -85,B 0,C 180,E1 -601.373,E2 -601.373} C_VEL
LIN {X 0,Y 601.4,Z 269.575,A -85,B 0,C 180,E1 -603.636,E2 -603.636} C_VEL
LIN {X 0,Y 601.416,Z 269.566,A -85,B 0,C 180,E1 -606.589,E2 -606.589} C_VEL
LIN {X 0,Y 601.421,Z 269.569,A -85,B 0,C 180,E1 -609.478,E2 -609.478} C_VEL
LIN {X 0,Y 601.39,Z 269.569,A -85,B 0,C 180,E1 -612.311,E2 -612.311} C_VEL
LIN {X 0,Y 601.416,Z 269.57,A -85,B 0,C 180,E1 -615.103,E2 -615.103} C_VEL
LIN {X 0,Y 601.402,Z 269.567,A -85,B 0,C 180,E1 -617.857,E2 -617.857} C_VEL
LIN {X 0,Y 601.401,Z 269.576,A -85,B 0,C 180,E1 -620.584,E2 -620.584} C_VEL
LIN {X 0,Y 601.386,Z 269.569,A -85,B 0,C 180,E1 -623.289,E2 -623.289} C_VEL
LIN {X 0,Y 601.397,Z 269.573,A -85,B 0,C 180,E1 -625.979,E2 -625.979} C_VEL
LIN {X 0,Y 601.374,Z 269.572,A -85,B 0,C 180,E1 -628.661,E2 -628.661} C_VEL
LIN {X 0,Y 601.358,Z 269.573,A -85,B 0,C 180,E1 -630.67,E2 -630.67} C_VEL
LIN {X 0,Y 601.392,Z 269.568,A -85,B 0,C 180,E1 -632.679,E2 -632.679} C_VEL
LIN {X 0,Y 601.403,Z 269.571,A -85,B 0,C 180,E1 -635.364,E2 -635.364} C_VEL
LIN {X 0,Y 601.426,Z 269.566,A -85,B 0,C 180,E1 -638.061,E2 -638.061} C_VEL
LIN {X 0,Y 601.4,Z 269.571,A -85,B 0,C 180,E1 -641.007,E2 -641.007} C_VEL
LIN {X 0,Y 601.418,Z 269.57,A -85,B 0,C 180,E1 -643.516,E2 -643.516} C_VEL
LIN {X 0,Y 601.42,Z 269.565,A -85,B 0,C 180,E1 -646.288,E2 -646.288} C_VEL
LIN {X 0,Y 601.41,Z 269.572,A -85,B 0,C 180,E1 -649.099,E2 -649.099} C_VEL
LIN {X 0,Y 601.407,Z 269.569,A -85,B 0,C 180,E1 -651.239,E2 -651.239} C_VEL
LIN {X 0,Y 601.445,Z 269.564,A -85,B 0,C 180,E1 -654.141,E2 -654.141} C_VEL
LIN {X 0,Y 601.448,Z 269.562,A -85,B 0,C 180,E1 -657.111,E2 -657.111} C_VEL
LIN {X 0,Y 601.416,Z 269.565,A -85,B 0,C 180,E1 -659.393,E2 -659.393} C_VEL
LIN {X 0,Y 601.407,Z 269.569,A -85,B 0,C 180,E1 -661.727,E2 -661.727} C_VEL
LIN {X 0,Y 601.424,Z 269.572,A -85,B 0,C 180,E1 -664.119,E2 -664.119} C_VEL
LIN {X 0,Y 601.405,Z 269.567,A -85,B 0,C 180,E1 -666.583,E2 -666.583} C_VEL
LIN {X 0,Y 601.44,Z 269.569,A -85,B 0,C 180,E1 -669.538,E2 -669.538} C_VEL
LIN {X 0,Y 601.396,Z 269.567,A -85,B 0,C 180,E1 -672.591,E2 -672.591} C_VEL
LIN {X 0,Y 601.39,Z 269.576,A -85,B 0,C 180,E1 -675.48,E2 -675.48} C_VEL
LIN {X 0,Y 601.405,Z 269.567,A -85,B 0,C 180,E1 -678.409,E2 -678.409} C_VEL
LIN {X 0,Y 601.392,Z 269.57,A -85,B 0,C 180,E1 -681.534,E2 -681.534} C_VEL
LIN {X 0,Y 601.378,Z 269.57,A -85,B 0,C 180,E1 -683.743,E2 -683.743} C_VEL
LIN {X 0,Y 601.402,Z 269.576,A -85,B 0,C 180,E1 -686.686,E2 -686.686} C_VEL
LIN {X 0,Y 601.385,Z 269.572,A -85,B 0,C 180,E1 -689.057,E2 -689.057} C_VEL
LIN {X 0,Y 601.419,Z 269.758,A -85,B 0,C 180,E1 -690.32,E2 -690.32} C_VEL
LIN {X 0,Y 601.389,Z 275.919,A -85,B 0,C 180,E1 -692.887,E2 -692.887} C_VEL
LIN {X 0,Y 601.37,Z 281.307,A -85,B 0,C 180,E1 -695.121,E2 -695.121} C_VEL
LIN {X 0,Y 601.344,Z 286.959,A -85,B 0,C 180,E1 -697.412,E2 -697.412} C_VEL
LIN {X 0,Y 601.36,Z 293.934,A -85,B 0,C 180,E1 -700.19,E2 -700.19} C_VEL
LIN {X 0,Y 601.322,Z 301.15,A -85,B 0,C 180,E1 -703.012,E2 -703.012} C_VEL
LIN {X 0,Y 601.348,Z 308.741,A -85,B 0,C 180,E1 -705.938,E2 -705.938} C_VEL
LIN {X 0,Y 601.312,Z 315.582,A -85,B 0,C 180,E1 -708.541,E2 -708.541} C_VEL
LIN {X 0,Y 601.325,Z 322.799,A -85,B 0,C 180,E1 -711.262,E2 -711.262} C_VEL
LIN {X 0,Y 601.332,Z 327.686,A -85,B 0,C 180,E1 -713.093,E2 -713.093} C_VEL
LIN {X 0,Y 601.428,Z 337.503,A -85,B 0,C 180,E1 -713.432,E2 -713.432} C_VEL
LIN {X 0,Y 601.412,Z 346.199,A -85,B 0,C 180,E1 -713.863,E2 -713.863} C_VEL
LIN {X 0,Y 601.376,Z 354.191,A -85,B 0,C 180,E1 -714.384,E2 -714.384} C_VEL
LIN {X 0,Y 601.374,Z 361.051,A -85,B 0,C 180,E1 -714.973,E2 -714.973} C_VEL
LIN {X 0,Y 601.362,Z 367.219,A -85,B 0,C 180,E1 -715.644,E2 -715.644} C_VEL
LIN {X 0,Y 601.374,Z 372.074,A -85,B 0,C 180,E1 -716.316,E2 -716.316} C_VEL
LIN {X 0,Y 601.379,Z 375.829,A -85,B 0,C 180,E1 -716.986,E2 -716.986} C_VEL
LIN {X 0,Y 601.345,Z 379.835,A -85,B 0,C 180,E1 -717.992,E2 -717.992} C_VEL
LIN {X 0,Y 601.347,Z 381.57,A -85,B 0,C 180,E1 -718.662,E2 -718.662} C_VEL
LIN {X 0,Y 601.339,Z 382.609,A -85,B 0,C 180,E1 -719.331,E2 -719.331} C_VEL
LIN {X 0,Y 601.336,Z 382.989,A -85,B 0,C 180,E1 -720.001,E2 -720.001} C_VEL
LIN {X 0,Y 601.339,Z 382.71,A -85,B 0,C 180,E1 -720.671,E2 -720.671} C_VEL
LIN {X 0,Y 601.349,Z 381.765,A -85,B 0,C 180,E1 -721.34,E2 -721.34} C_VEL
LIN {X 0,Y 601.345,Z 380.126,A -85,B 0,C 180,E1 -722.01,E2 -722.01} C_VEL
LIN {X 0,Y 601.332,Z 377.743,A -85,B 0,C 180,E1 -722.68,E2 -722.68} C_VEL
LIN {X 0,Y 601.375,Z 372.615,A -85,B 0,C 180,E1 -723.686,E2 -723.686} C_VEL
LIN {X 0,Y 601.378,Z 366.544,A -85,B 0,C 180,E1 -724.525,E2 -724.525} C_VEL
LIN {X 0,Y 601.346,Z 360.24,A -85,B 0,C 180,E1 -725.198,E2 -725.198} C_VEL
LIN {X 0,Y 601.385,Z 353.076,A -85,B 0,C 180,E1 -725.786,E2 -725.786} C_VEL
LIN {X 0,Y 601.4,Z 344.658,A -85,B 0,C 180,E1 -726.314,E2 -726.314} C_VEL
LIN {X 0,Y 601.428,Z 335.077,A -85,B 0,C 180,E1 -726.754,E2 -726.754} C_VEL
LIN {X 0,Y 601.333,Z 327.659,A -85,B 0,C 180,E1 -727.008,E2 -727.008} C_VEL
LIN {X 0,Y 601.32,Z 321.23,A -85,B 0,C 180,E1 -729.418,E2 -729.418} C_VEL
LIN {X 0,Y 601.352,Z 314.011,A -85,B 0,C 180,E1 -732.145,E2 -732.145} C_VEL
LIN {X 0,Y 601.349,Z 306.792,A -85,B 0,C 180,E1 -734.9,E2 -734.9} C_VEL
LIN {X 0,Y 601.354,Z 299.572,A -85,B 0,C 180,E1 -737.69,E2 -737.69} C_VEL
LIN {X 0,Y 601.366,Z 294.158,A -85,B 0,C 180,E1 -739.811,E2 -739.811} C_VEL
LIN {X 0,Y 601.356,Z 286.938,A -85,B 0,C 180,E1 -742.686,E2 -742.686} C_VEL
LIN {X 0,Y 601.399,Z 279.718,A -85,B 0,C 180,E1 -745.62,E2 -745.62} C_VEL
LIN {X 0,Y 601.386,Z 274.315,A -85,B 0,C 180,E1 -747.87,E2 -747.87} C_VEL
LIN {X 0,Y 601.412,Z 269.573,A -85,B 0,C 180,E1 -749.825,E2 -749.825} C_VEL
LIN {X 0,Y 601.423,Z 269.574,A -85,B 0,C 180,E1 -752.715,E2 -752.715} C_VEL
LIN {X 0,Y 601.408,Z 269.573,A -85,B 0,C 180,E1 -755.113,E2 -755.113} C_VEL
LIN {X 0,Y 601.441,Z 269.569,A -85,B 0,C 180,E1 -757.419,E2 -757.419} C_VEL
LIN {X 0,Y 601.407,Z 269.575,A -85,B 0,C 180,E1 -759.996,E2 -759.996} C_VEL
LIN {X 0,Y 601.415,Z 269.572,A -85,B 0,C 180,E1 -762.671,E2 -762.671} C_VEL
LIN {X 0,Y 601.403,Z 269.575,A -85,B 0,C 180,E1 -765.48,E2 -765.48} C_VEL
LIN {X 0,Y 601.428,Z 269.573,A -85,B 0,C 180,E1 -768.407,E2 -768.407} C_VEL
LIN {X 0,Y 601.413,Z 269.573,A -85,B 0,C 180,E1 -770.873,E2 -770.873} C_VEL
LIN {X 0,Y 601.405,Z 269.574,A -85,B 0,C 180,E1 -773.417,E2 -773.417} C_VEL
LIN {X 0,Y 601.435,Z 269.571,A -85,B 0,C 180,E1 -776.065,E2 -776.065} C_VEL
LIN {X 0,Y 601.424,Z 269.571,A -85,B 0,C 180,E1 -778.545,E2 -778.545} C_VEL
LIN {X 0,Y 601.428,Z 269.572,A -85,B 0,C 180,E1 -781.373,E2 -781.373} C_VEL
LIN {X 0,Y 601.437,Z 269.694,A -85,B 0,C 180,E1 -782.201,E2 -782.201} C_VEL
LIN {X 0,Y 601.781,Z 273.898,A -85,B 0,C 180,E1 -782.905,E2 -782.905} C_VEL
LIN {X 0,Y 601.661,Z 291.057,A -85,B 0,C 180,E1 -785.661,E2 -785.661} C_VEL
LIN {X 0,Y 601.595,Z 308.515,A -85,B 0,C 180,E1 -788.408,E2 -788.408} C_VEL
LIN {X 0,Y 601.535,Z 324.67,A -85,B 0,C 180,E1 -790.905,E2 -790.905} C_VEL
LIN {X 0,Y 601.506,Z 343.133,A -85,B 0,C 180,E1 -793.715,E2 -793.715} C_VEL
LIN {X 0,Y 601.445,Z 361.595,A -85,B 0,C 180,E1 -796.485,E2 -796.485} C_VEL
LIN {X 0,Y 601.438,Z 372.198,A -85,B 0,C 180,E1 -798.04,E2 -798.04} C_VEL
LIN {X 0,Y 601.58,Z 385.435,A -85,B 0,C 180,E1 -798.267,E2 -798.267} C_VEL
LIN {X 0,Y 601.554,Z 398.236,A -85,B 0,C 180,E1 -798.622,E2 -798.622} C_VEL
LIN {X 0,Y 601.538,Z 409.964,A -85,B 0,C 180,E1 -799.077,E2 -799.077} C_VEL
LIN {X 0,Y 601.488,Z 421.327,A -85,B 0,C 180,E1 -799.651,E2 -799.651} C_VEL
LIN {X 0,Y 601.469,Z 431.93,A -85,B 0,C 180,E1 -800.33,E2 -800.33} C_VEL
LIN {X 0,Y 601.435,Z 441.598,A -85,B 0,C 180,E1 -801.093,E2 -801.093} C_VEL
LIN {X 0,Y 601.407,Z 450.413,A -85,B 0,C 180,E1 -801.939,E2 -801.939} C_VEL
LIN {X 0,Y 601.388,Z 457.69,A -85,B 0,C 180,E1 -802.783,E2 -802.783} C_VEL
LIN {X 0,Y 601.375,Z 464.774,A -85,B 0,C 180,E1 -803.782,E2 -803.782} C_VEL
LIN {X 0,Y 601.373,Z 469.68,A -85,B 0,C 180,E1 -804.635,E2 -804.635} C_VEL
LIN {X 0,Y 601.354,Z 474.371,A -85,B 0,C 180,E1 -805.643,E2 -805.643} C_VEL
LIN {X 0,Y 601.344,Z 477.956,A -85,B 0,C 180,E1 -806.65,E2 -806.65} C_VEL
LIN {X 0,Y 601.325,Z 479.809,A -85,B 0,C 180,E1 -807.32,E2 -807.32} C_VEL
LIN {X 0,Y 601.343,Z 481.202,A -85,B 0,C 180,E1 -807.991,E2 -807.991} C_VEL
LIN {X 0,Y 601.339,Z 482.784,A -85,B 0,C 180,E1 -809.33,E2 -809.33} C_VEL
LIN {X 0,Y 601.335,Z 483,A -85,B 0,C 180,E1 -810,E2 -810} C_VEL
LIN {X 0,Y 601.347,Z 482.184,A -85,B 0,C 180,E1 -811.339,E2 -811.339} C_VEL
LIN {X 0,Y 601.343,Z 481.201,A -85,B 0,C 180,E1 -812.009,E2 -812.009} C_VEL
LIN {X 0,Y 601.325,Z 479.809,A -85,B 0,C 180,E1 -812.68,E2 -812.68} C_VEL
LIN {X 0,Y 601.368,Z 476.896,A -85,B 0,C 180,E1 -813.685,E2 -813.685} C_VEL
LIN {X 0,Y 601.336,Z 472.95,A -85,B 0,C 180,E1 -814.693,E2 -814.693} C_VEL
LIN {X 0,Y 601.373,Z 466.877,A -85,B 0,C 180,E1 -815.869,E2 -815.869} C_VEL
LIN {X 0,Y 601.382,Z 460.235,A -85,B 0,C 180,E1 -816.88,E2 -816.88} C_VEL
LIN {X 0,Y 601.4,Z 451.989,A -85,B 0,C 180,E1 -817.892,E2 -817.892} C_VEL
LIN {X 0,Y 601.436,Z 443.536,A -85,B 0,C 180,E1 -818.738,E2 -818.738} C_VEL
LIN {X 0,Y 601.45,Z 433.091,A -85,B 0,C 180,E1 -819.585,E2 -819.585} C_VEL
LIN {X 0,Y 601.473,Z 422.756,A -85,B 0,C 180,E1 -820.264,E2 -820.264} C_VEL
LIN {X 0,Y 601.534,Z 410.645,A -85,B 0,C 180,E1 -820.894,E2 -820.894} C_VEL
LIN {X 0,Y 601.554,Z 398.226,A -85,B 0,C 180,E1 -821.378,E2 -821.378} C_VEL
LIN {X 0,Y 601.582,Z 385.437,A -85,B 0,C 180,E1 -821.733,E2 -821.733} C_VEL
LIN {X 0,Y 601.421,Z 371.981,A -85,B 0,C 180,E1 -821.971,E2 -821.971} C_VEL
LIN {X 0,Y 601.444,Z 353.518,A -85,B 0,C 180,E1 -824.723,E2 -824.723} C_VEL
LIN {X 0,Y 601.518,Z 335.055,A -85,B 0,C 180,E1 -827.509,E2 -827.509} C_VEL
LIN {X 0,Y 601.561,Z 316.593,A -85,B 0,C 180,E1 -830.339,E2 -830.339} C_VEL
LIN {X 0,Y 601.634,Z 299.284,A -85,B 0,C 180,E1 -833.037,E2 -833.037} C_VEL
LIN {X 0,Y 601.731,Z 281.11,A -85,B 0,C 180,E1 -835.929,E2 -835.929} C_VEL
LIN {X 0,Y 601.706,Z 270.927,A -85,B 0,C 180,E1 -837.584,E2 -837.584} C_VEL
LIN {X 0,Y 601.424,Z 269.573,A -85,B 0,C 180,E1 -837.834,E2 -837.834} C_VEL
LIN {X 0,Y 601.433,Z 269.571,A -85,B 0,C 180,E1 -840.164,E2 -840.164} C_VEL
LIN {X 0,Y 601.419,Z 269.571,A -85,B 0,C 180,E1 -842.714,E2 -842.714} C_VEL
LIN {X 0,Y 601.392,Z 269.576,A -85,B 0,C 180,E1 -845.111,E2 -845.111} C_VEL
LIN {X 0,Y 601.439,Z 269.572,A -85,B 0,C 180,E1 -847.419,E2 -847.419} C_VEL
LIN {X 0,Y 601.416,Z 269.572,A -85,B 0,C 180,E1 -849.995,E2 -849.995} C_VEL
LIN {X 0,Y 601.412,Z 269.574,A -85,B 0,C 180,E1 -852.67,E2 -852.67} C_VEL
LIN {X 0,Y 601.432,Z 269.57,A -85,B 0,C 180,E1 -855.482,E2 -855.482} C_VEL
LIN {X 0,Y 601.426,Z 269.571,A -85,B 0,C 180,E1 -858.407,E2 -858.407} C_VEL
LIN {X 0,Y 601.436,Z 269.569,A -85,B 0,C 180,E1 -860.875,E2 -860.875} C_VEL
LIN {X 0,Y 601.408,Z 269.576,A -85,B 0,C 180,E1 -863.417,E2 -863.417} C_VEL
LIN {X 0,Y 601.421,Z 269.571,A -85,B 0,C 180,E1 -866.066,E2 -866.066} C_VEL
LIN {X 0,Y 601.423,Z 269.573,A -85,B 0,C 180,E1 -868.545,E2 -868.545} C_VEL
LIN {X 0,Y 601.365,Z 269.696,A -85,B 0,C 180,E1 -870.816,E2 -870.816} C_VEL
LIN {X 0,Y 601.357,Z 275.607,A -85,B 0,C 180,E1 -872.884,E2 -872.884} C_VEL
LIN {X 0,Y 601.34,Z 281.303,A -85,B 0,C 180,E1 -875.118,E2 -875.118} C_VEL
LIN {X 0,Y 601.35,Z 286.954,A -85,B 0,C 180,E1 -877.41,E2 -877.41} C_VEL
LIN {X 0,Y 601.361,Z 293.93,A -85,B 0,C 180,E1 -880.188,E2 -880.188} C_VEL
LIN {X 0,Y 601.324,Z 301.145,A -85,B 0,C 180,E1 -883.01,E2 -883.01} C_VEL
LIN {X 0,Y 601.352,Z 308.738,A -85,B 0,C 180,E1 -885.936,E2 -885.936} C_VEL
LIN {X 0,Y 601.311,Z 315.578,A -85,B 0,C 180,E1 -888.539,E2 -888.539} C_VEL
LIN {X 0,Y 601.325,Z 322.794,A -85,B 0,C 180,E1 -891.26,E2 -891.26} C_VEL
LIN {X 0,Y 601.332,Z 327.684,A -85,B 0,C 180,E1 -893.092,E2 -893.092} C_VEL
LIN {X 0,Y 601.433,Z 337.861,A -85,B 0,C 180,E1 -893.447,E2 -893.447} C_VEL
LIN {X 0,Y 601.412,Z 346.195,A -85,B 0,C 180,E1 -893.862,E2 -893.862} C_VEL
LIN {X 0,Y 601.376,Z 354.172,A -85,B 0,C 180,E1 -894.382,E2 -894.382} C_VEL
LIN {X 0,Y 601.374,Z 361.033,A -85,B 0,C 180,E1 -894.971,E2 -894.971} C_VEL
LIN {X 0,Y 601.362,Z 367.21,A -85,B 0,C 180,E1 -895.643,E2 -895.643} C_VEL
LIN {X 0,Y 601.374,Z 372.063,A -85,B 0,C 180,E1 -896.314,E2 -896.314} C_VEL
LIN {X 0,Y 601.379,Z 375.82,A -85,B 0,C 180,E1 -896.985,E2 -896.985} C_VEL
LIN {X 0,Y 601.345,Z 379.826,A -85,B 0,C 180,E1 -897.99,E2 -897.99} C_VEL
LIN {X 0,Y 601.348,Z 381.567,A -85,B 0,C 180,E1 -898.66,E2 -898.66} C_VEL
LIN {X 0,Y 601.34,Z 382.614,A -85,B 0,C 180,E1 -899.329,E2 -899.329} C_VEL
LIN {X 0,Y 601.336,Z 382.995,A -85,B 0,C 180,E1 -899.999,E2 -899.999} C_VEL
LIN {X 0,Y 601.339,Z 382.715,A -85,B 0,C 180,E1 -900.669,E2 -900.669} C_VEL
LIN {X 0,Y 601.349,Z 381.768,A -85,B 0,C 180,E1 -901.338,E2 -901.338} C_VEL
LIN {X 0,Y 601.345,Z 380.128,A -85,B 0,C 180,E1 -902.008,E2 -902.008} C_VEL
LIN {X 0,Y 601.38,Z 376.236,A -85,B 0,C 180,E1 -903.014,E2 -903.014} C_VEL
LIN {X 0,Y 601.38,Z 371.559,A -85,B 0,C 180,E1 -903.852,E2 -903.852} C_VEL
LIN {X 0,Y 601.379,Z 366.565,A -85,B 0,C 180,E1 -904.523,E2 -904.523} C_VEL
LIN {X 0,Y 601.346,Z 360.261,A -85,B 0,C 180,E1 -905.196,E2 -905.196} C_VEL
LIN {X 0,Y 601.384,Z 353.11,A -85,B 0,C 180,E1 -905.784,E2 -905.784} C_VEL
LIN {X 0,Y 601.4,Z 344.685,A -85,B 0,C 180,E1 -906.314,E2 -906.314} C_VEL
LIN {X 0,Y 601.426,Z 335.125,A -85,B 0,C 180,E1 -906.752,E2 -906.752} C_VEL
LIN {X 0,Y 601.333,Z 327.663,A -85,B 0,C 180,E1 -907.006,E2 -907.006} C_VEL
LIN {X 0,Y 601.32,Z 321.234,A -85,B 0,C 180,E1 -909.416,E2 -909.416} C_VEL
LIN {X 0,Y 601.329,Z 314.489,A -85,B 0,C 180,E1 -911.964,E2 -911.964} C_VEL
LIN {X 0,Y 600.695,Z 313.094,A -85,B 0,C 180,E1 -912.507,E2 -912.507} C_VEL
LIN {X 0,Y 597.835,Z 310.944,A -85,B 0,C 180,E1 -913.391,E2 -913.391} C_VEL
LIN {X 0,Y 595.397,Z 309.244,A -85,B 0,C 180,E1 -914.102,E2 -914.102} C_VEL
LIN {X 0,Y 594.348,Z 307.895,A -85,B 0,C 180,E1 -914.65,E2 -914.65} C_VEL
LIN {X 0,Y 594.263,Z 307.423,A -85,B 0,C 180,E1 -914.836,E2 -914.836} C_VEL
LIN {X 0,Y 594.27,Z 301.38,A -85,B 0,C 180,E1 -917.196,E2 -917.196} C_VEL
LIN {X 0,Y 594.28,Z 295.966,A -85,B 0,C 180,E1 -919.336,E2 -919.336} C_VEL
LIN {X 0,Y 594.29,Z 288.746,A -85,B 0,C 180,E1 -922.235,E2 -922.235} C_VEL
LIN {X 0,Y 594.323,Z 281.5,A -85,B 0,C 180,E1 -925.194,E2 -925.194} C_VEL
LIN {X 0,Y 594.324,Z 273.953,A -85,B 0,C 180,E1 -928.228,E2 -928.228} C_VEL
LIN {X 0,Y 594.36,Z 270.45,A -85,B 0,C 180,E1 -929.678,E2 -929.678} C_VEL
LIN {X 0,Y 594.329,Z 270.448,A -85,B 0,C 180,E1 -932.148,E2 -932.148} C_VEL
LIN {X 0,Y 594.352,Z 270.446,A -85,B 0,C 180,E1 -934.58,E2 -934.58} C_VEL
LIN {X 0,Y 594.376,Z 270.443,A -85,B 0,C 180,E1 -937.606,E2 -937.606} C_VEL
LIN {X 0,Y 594.353,Z 270.45,A -85,B 0,C 180,E1 -940.567,E2 -940.567} C_VEL
LIN {X 0,Y 594.344,Z 270.447,A -85,B 0,C 180,E1 -943.3,E2 -943.3} C_VEL
LIN {X 0,Y 594.352,Z 270.449,A -85,B 0,C 180,E1 -946.16,E2 -946.16} C_VEL
LIN {X 0,Y 594.371,Z 270.443,A -85,B 0,C 180,E1 -949.177,E2 -949.177} C_VEL
LIN {X 0,Y 594.377,Z 270.45,A -85,B 0,C 180,E1 -952.058,E2 -952.058} C_VEL
LIN {X 0,Y 594.374,Z 270.444,A -85,B 0,C 180,E1 -954.671,E2 -954.671} C_VEL
LIN {X 0,Y 594.371,Z 270.443,A -85,B 0,C 180,E1 -957.087,E2 -957.087} C_VEL
LIN {X 0,Y 594.392,Z 270.449,A -85,B 0,C 180,E1 -959.668,E2 -959.668} C_VEL
LIN {X 0,Y 594.381,Z 270.441,A -85,B 0,C 180,E1 -962.539,E2 -962.539} C_VEL
LIN {X 0,Y 594.37,Z 270.444,A -85,B 0,C 180,E1 -964.807,E2 -964.807} C_VEL
LIN {X 0,Y 594.356,Z 270.454,A -85,B 0,C 180,E1 -967.263,E2 -967.263} C_VEL
LIN {X 0,Y 594.365,Z 270.444,A -85,B 0,C 180,E1 -969.946,E2 -969.946} C_VEL
LIN {X 0,Y 594.379,Z 270.449,A -85,B 0,C 180,E1 -972.806,E2 -972.806} C_VEL
LIN {X 0,Y 594.376,Z 270.442,A -85,B 0,C 180,E1 -975.826,E2 -975.826} C_VEL
LIN {X 0,Y 594.382,Z 270.447,A -85,B 0,C 180,E1 -978.404,E2 -978.404} C_VEL
LIN {X 0,Y 594.352,Z 270.446,A -85,B 0,C 180,E1 -981.157,E2 -981.157} C_VEL
LIN {X 0,Y 594.374,Z 270.445,A -85,B 0,C 180,E1 -983.891,E2 -983.891} C_VEL
LIN {X 0,Y 594.318,Z 270.452,A -85,B 0,C 180,E1 -986.61,E2 -986.61} C_VEL
LIN {X 0,Y 594.332,Z 270.449,A -85,B 0,C 180,E1 -988.645,E2 -988.645} C_VEL
LIN {X 0,Y 594.313,Z 270.45,A -85,B 0,C 180,E1 -990.678,E2 -990.678} C_VEL
LIN {X 0,Y 594.36,Z 270.444,A -85,B 0,C 180,E1 -992.711,E2 -992.711} C_VEL
LIN {X 0,Y 594.372,Z 270.448,A -85,B 0,C 180,E1 -995.428,E2 -995.428} C_VEL
LIN {X 0,Y 594.397,Z 270.441,A -85,B 0,C 180,E1 -998.157,E2 -998.157} C_VEL
LIN {X 0,Y 594.365,Z 270.448,A -85,B 0,C 180,E1 -1001.069,E2 -1001.069} C_VEL
LIN {X 0,Y 594.378,Z 270.444,A -85,B 0,C 180,E1 -1003.679,E2 -1003.679} C_VEL
LIN {X 0,Y 594.376,Z 270.447,A -85,B 0,C 180,E1 -1006.718,E2 -1006.718} C_VEL
LIN {X 0,Y 594.359,Z 270.447,A -85,B 0,C 180,E1 -1009.335,E2 -1009.335} C_VEL
LIN {X 0,Y 594.363,Z 270.444,A -85,B 0,C 180,E1 -1011.504,E2 -1011.504} C_VEL
LIN {X 0,Y 594.378,Z 270.449,A -85,B 0,C 180,E1 -1014.447,E2 -1014.447} C_VEL
LIN {X 0,Y 594.381,Z 270.447,A -85,B 0,C 180,E1 -1016.7,E2 -1016.7} C_VEL
LIN {X 0,Y 594.377,Z 270.443,A -85,B 0,C 180,E1 -1018.999,E2 -1018.999} C_VEL
LIN {X 0,Y 594.385,Z 270.443,A -85,B 0,C 180,E1 -1021.646,E2 -1021.646} C_VEL
LIN {X 0,Y 594.384,Z 270.443,A -85,B 0,C 180,E1 -1024.58,E2 -1024.58} C_VEL
LIN {X 0,Y 594.379,Z 270.442,A -85,B 0,C 180,E1 -1027.087,E2 -1027.087} C_VEL
LIN {X 0,Y 594.373,Z 270.451,A -85,B 0,C 180,E1 -1029.776,E2 -1029.776} C_VEL
LIN {X 0,Y 594.354,Z 270.445,A -85,B 0,C 180,E1 -1032.377,E2 -1032.377} C_VEL
LIN {X 0,Y 594.348,Z 270.452,A -85,B 0,C 180,E1 -1035.193,E2 -1035.193} C_VEL
LIN {X 0,Y 594.36,Z 270.444,A -85,B 0,C 180,E1 -1038.154,E2 -1038.154} C_VEL
LIN {X 0,Y 594.361,Z 270.451,A -85,B 0,C 180,E1 -1041.195,E2 -1041.195} C_VEL
LIN {X 0,Y 594.332,Z 270.447,A -85,B 0,C 180,E1 -1043.756,E2 -1043.756} C_VEL
LIN {X 0,Y 594.343,Z 270.448,A -85,B 0,C 180,E1 -1046.238,E2 -1046.238} C_VEL
LIN {X 0,Y 594.354,Z 270.454,A -85,B 0,C 180,E1 -1048.65,E2 -1048.65} C_VEL
LIN {X 0,Y 594.383,Z 270.551,A -85,B 0,C 180,E1 -1050.274,E2 -1050.274} C_VEL
LIN {X 0,Y 594.372,Z 276,A -85,B 0,C 180,E1 -1052.54,E2 -1052.54} C_VEL
LIN {X 0,Y 594.312,Z 281.3,A -85,B 0,C 180,E1 -1054.805,E2 -1054.805} C_VEL
LIN {X 0,Y 594.287,Z 288.524,A -85,B 0,C 180,E1 -1057.765,E2 -1057.765} C_VEL
LIN {X 0,Y 594.276,Z 295.74,A -85,B 0,C 180,E1 -1060.664,E2 -1060.664} C_VEL
LIN {X 0,Y 594.258,Z 302.956,A -85,B 0,C 180,E1 -1063.512,E2 -1063.512} C_VEL
LIN {X 0,Y 594.245,Z 310.172,A -85,B 0,C 180,E1 -1066.319,E2 -1066.319} C_VEL
LIN {X 0,Y 594.238,Z 317.388,A -85,B 0,C 180,E1 -1069.093,E2 -1069.093} C_VEL
LIN {X 0,Y 594.255,Z 324.605,A -85,B 0,C 180,E1 -1071.842,E2 -1071.842} C_VEL
LIN {X 0,Y 594.239,Z 327.706,A -85,B 0,C 180,E1 -1073.017,E2 -1073.017} C_VEL
LIN {X 0,Y 594.367,Z 337.139,A -85,B 0,C 180,E1 -1073.338,E2 -1073.338} C_VEL
LIN {X 0,Y 594.359,Z 344.815,A -85,B 0,C 180,E1 -1073.71,E2 -1073.71} C_VEL
LIN {X 0,Y 594.315,Z 353.017,A -85,B 0,C 180,E1 -1074.232,E2 -1074.232} C_VEL
LIN {X 0,Y 594.307,Z 361.063,A -85,B 0,C 180,E1 -1074.913,E2 -1074.913} C_VEL
LIN {X 0,Y 594.286,Z 367.224,A -85,B 0,C 180,E1 -1075.592,E2 -1075.592} C_VEL
LIN {X 0,Y 594.3,Z 372.075,A -85,B 0,C 180,E1 -1076.272,E2 -1076.272} C_VEL
LIN {X 0,Y 594.278,Z 375.832,A -85,B 0,C 180,E1 -1076.95,E2 -1076.95} C_VEL
LIN {X 0,Y 594.245,Z 379.841,A -85,B 0,C 180,E1 -1077.968,E2 -1077.968} C_VEL
LIN {X 0,Y 594.247,Z 381.571,A -85,B 0,C 180,E1 -1078.646,E2 -1078.646} C_VEL
LIN {X 0,Y 594.24,Z 382.603,A -85,B 0,C 180,E1 -1079.323,E2 -1079.323} C_VEL
LIN {X 0,Y 594.236,Z 382.981,A -85,B 0,C 180,E1 -1080.001,E2 -1080.001} C_VEL
LIN {X 0,Y 594.239,Z 382.706,A -85,B 0,C 180,E1 -1080.679,E2 -1080.679} C_VEL
LIN {X 0,Y 594.249,Z 381.764,A -85,B 0,C 180,E1 -1081.356,E2 -1081.356} C_VEL
LIN {X 0,Y 594.245,Z 380.125,A -85,B 0,C 180,E1 -1082.034,E2 -1082.034} C_VEL
LIN {X 0,Y 594.279,Z 376.235,A -85,B 0,C 180,E1 -1083.051,E2 -1083.051} C_VEL
LIN {X 0,Y 594.301,Z 371.531,A -85,B 0,C 180,E1 -1083.9,E2 -1083.9} C_VEL
LIN {X 0,Y 594.31,Z 366.54,A -85,B 0,C 180,E1 -1084.579,E2 -1084.579} C_VEL
LIN {X 0,Y 594.264,Z 360.231,A -85,B 0,C 180,E1 -1085.26,E2 -1085.26} C_VEL
LIN {X 0,Y 594.326,Z 353.06,A -85,B 0,C 180,E1 -1085.855,E2 -1085.855} C_VEL
LIN {X 0,Y 594.357,Z 345.394,A -85,B 0,C 180,E1 -1086.347,E2 -1086.347} C_VEL
LIN {X 0,Y 594.369,Z 336.19,A -85,B 0,C 180,E1 -1086.792,E2 -1086.792} C_VEL
LIN {X 0,Y 594.243,Z 327.657,A -85,B 0,C 180,E1 -1087.092,E2 -1087.092} C_VEL
LIN {X 0,Y 594.244,Z 321.228,A -85,B 0,C 180,E1 -1089.531,E2 -1089.531} C_VEL
LIN {X 0,Y 594.248,Z 314.009,A -85,B 0,C 180,E1 -1092.292,E2 -1092.292} C_VEL
LIN {X 0,Y 594.266,Z 306.79,A -85,B 0,C 180,E1 -1095.081,E2 -1095.081} C_VEL
LIN {X 0,Y 594.265,Z 299.571,A -85,B 0,C 180,E1 -1097.908,E2 -1097.908} C_VEL
LIN {X 0,Y 594.272,Z 294.156,A -85,B 0,C 180,E1 -1100.058,E2 -1100.058} C_VEL
LIN {X 0,Y 594.293,Z 286.936,A -85,B 0,C 180,E1 -1102.971,E2 -1102.971} C_VEL
LIN {X 0,Y 594.35,Z 281.662,A -85,B 0,C 180,E1 -1105.195,E2 -1105.195} C_VEL
LIN {X 0,Y 594.348,Z 276.076,A -85,B 0,C 180,E1 -1107.519,E2 -1107.519} C_VEL
LIN {X 0,Y 594.369,Z 270.45,A -85,B 0,C 180,E1 -1109.864,E2 -1109.864} C_VEL
LIN {X 0,Y 594.368,Z 270.45,A -85,B 0,C 180,E1 -1112.148,E2 -1112.148} C_VEL
LIN {X 0,Y 594.39,Z 270.448,A -85,B 0,C 180,E1 -1114.58,E2 -1114.58} C_VEL
LIN {X 0,Y 594.395,Z 270.447,A -85,B 0,C 180,E1 -1117.609,E2 -1117.609} C_VEL
LIN {X 0,Y 594.372,Z 270.449,A -85,B 0,C 180,E1 -1120.567,E2 -1120.567} C_VEL
LIN {X 0,Y 594.372,Z 270.451,A -85,B 0,C 180,E1 -1123.3,E2 -1123.3} C_VEL
LIN {X 0,Y 594.365,Z 270.451,A -85,B 0,C 180,E1 -1126.161,E2 -1126.161} C_VEL
LIN {X 0,Y 594.385,Z 270.45,A -85,B 0,C 180,E1 -1128.536,E2 -1128.536} C_VEL
LIN {X 0,Y 594.379,Z 270.449,A -85,B 0,C 180,E1 -1131.297,E2 -1131.297} C_VEL
LIN {X 0,Y 594.355,Z 270.454,A -85,B 0,C 180,E1 -1133.755,E2 -1133.755} C_VEL
LIN {X 0,Y 594.379,Z 270.449,A -85,B 0,C 180,E1 -1136.239,E2 -1136.239} C_VEL
LIN {X 0,Y 594.375,Z 270.45,A -85,B 0,C 180,E1 -1138.65,E2 -1138.65} C_VEL
LIN {X 0,Y 594.386,Z 270.45,A -85,B 0,C 180,E1 -1141.042,E2 -1141.042} C_VEL
LIN {X 0,Y 594.405,Z 270.567,A -85,B 0,C 180,E1 -1141.972,E2 -1141.972} C_VEL
LIN {X 0,Y 594.895,Z 273.898,A -85,B 0,C 180,E1 -1142.565,E2 -1142.565} C_VEL
LIN {X 0,Y 594.787,Z 290.283,A -85,B 0,C 180,E1 -1145.236,E2 -1145.236} C_VEL
LIN {X 0,Y 594.654,Z 308.515,A -85,B 0,C 180,E1 -1148.143,E2 -1148.143} C_VEL
LIN {X 0,Y 594.573,Z 326.166,A -85,B 0,C 180,E1 -1150.905,E2 -1150.905} C_VEL
LIN {X 0,Y 594.495,Z 344.287,A -85,B 0,C 180,E1 -1153.694,E2 -1153.694} C_VEL
LIN {X 0,Y 594.425,Z 363.903,A -85,B 0,C 180,E1 -1156.67,E2 -1156.67} C_VEL
LIN {X 0,Y 594.397,Z 372.198,A -85,B 0,C 180,E1 -1157.896,E2 -1157.896} C_VEL
LIN {X 0,Y 594.661,Z 380.084,A -85,B 0,C 180,E1 -1158.02,E2 -1158.02} C_VEL
LIN {X 0,Y 594.62,Z 393.732,A -85,B 0,C 180,E1 -1158.344,E2 -1158.344} C_VEL
LIN {X 0,Y 594.563,Z 406.27,A -85,B 0,C 180,E1 -1158.786,E2 -1158.786} C_VEL
LIN {X 0,Y 594.515,Z 418.209,A -85,B 0,C 180,E1 -1159.356,E2 -1159.356} C_VEL
LIN {X 0,Y 594.473,Z 429.477,A -85,B 0,C 180,E1 -1160.043,E2 -1160.043} C_VEL
LIN {X 0,Y 594.406,Z 439.646,A -85,B 0,C 180,E1 -1160.815,E2 -1160.815} C_VEL
LIN {X 0,Y 594.373,Z 448.787,A -85,B 0,C 180,E1 -1161.672,E2 -1161.672} C_VEL
LIN {X 0,Y 594.317,Z 457.69,A -85,B 0,C 180,E1 -1162.697,E2 -1162.697} C_VEL
LIN {X 0,Y 594.281,Z 464.171,A -85,B 0,C 180,E1 -1163.615,E2 -1163.615} C_VEL
LIN {X 0,Y 594.289,Z 469.68,A -85,B 0,C 180,E1 -1164.571,E2 -1164.571} C_VEL
LIN {X 0,Y 594.27,Z 474.371,A -85,B 0,C 180,E1 -1165.591,E2 -1165.591} C_VEL
LIN {X 0,Y 594.267,Z 477.957,A -85,B 0,C 180,E1 -1166.61,E2 -1166.61} C_VEL
LIN {X 0,Y 594.226,Z 479.809,A -85,B 0,C 180,E1 -1167.288,E2 -1167.288} C_VEL
LIN {X 0,Y 594.242,Z 481.202,A -85,B 0,C 180,E1 -1167.967,E2 -1167.967} C_VEL
LIN {X 0,Y 594.239,Z 482.784,A -85,B 0,C 180,E1 -1169.322,E2 -1169.322} C_VEL
LIN {X 0,Y 594.236,Z 483,A -85,B 0,C 180,E1 -1170,E2 -1170} C_VEL
LIN {X 0,Y 594.247,Z 482.184,A -85,B 0,C 180,E1 -1171.355,E2 -1171.355} C_VEL
LIN {X 0,Y 594.242,Z 481.201,A -85,B 0,C 180,E1 -1172.033,E2 -1172.033} C_VEL
LIN {X 0,Y 594.226,Z 479.809,A -85,B 0,C 180,E1 -1172.712,E2 -1172.712} C_VEL
LIN {X 0,Y 594.289,Z 476.896,A -85,B 0,C 180,E1 -1173.729,E2 -1173.729} C_VEL
LIN {X 0,Y 594.241,Z 472.95,A -85,B 0,C 180,E1 -1174.749,E2 -1174.749} C_VEL
LIN {X 0,Y 594.305,Z 466.877,A -85,B 0,C 180,E1 -1175.939,E2 -1175.939} C_VEL
LIN {X 0,Y 594.308,Z 460.236,A -85,B 0,C 180,E1 -1176.962,E2 -1176.962} C_VEL
LIN {X 0,Y 594.359,Z 451.99,A -85,B 0,C 180,E1 -1177.986,E2 -1177.986} C_VEL
LIN {X 0,Y 594.382,Z 443.536,A -85,B 0,C 180,E1 -1178.842,E2 -1178.842} C_VEL
LIN {X 0,Y 594.433,Z 433.093,A -85,B 0,C 180,E1 -1179.699,E2 -1179.699} C_VEL
LIN {X 0,Y 594.489,Z 422.757,A -85,B 0,C 180,E1 -1180.386,E2 -1180.386} C_VEL
LIN {X 0,Y 594.553,Z 411.779,A -85,B 0,C 180,E1 -1180.971,E2 -1180.971} C_VEL
LIN {X 0,Y 594.578,Z 399.728,A -85,B 0,C 180,E1 -1181.464,E2 -1181.464} C_VEL
LIN {X 0,Y 594.634,Z 386.351,A -85,B 0,C 180,E1 -1181.85,E2 -1181.85} C_VEL
LIN {X 0,Y 594.509,Z 373.079,A -85,B 0,C 180,E1 -1182.091,E2 -1182.091} C_VEL
LIN {X 0,Y 594.382,Z 371.981,A -85,B 0,C 180,E1 -1182.115,E2 -1182.115} C_VEL
LIN {X 0,Y 594.437,Z 353.518,A -85,B 0,C 180,E1 -1184.901,E2 -1184.901} C_VEL
LIN {X 0,Y 594.533,Z 335.055,A -85,B 0,C 180,E1 -1187.722,E2 -1187.722} C_VEL
LIN {X 0,Y 594.625,Z 316.593,A -85,B 0,C 180,E1 -1190.587,E2 -1190.587} C_VEL
LIN {X 0,Y 594.752,Z 298.13,A -85,B 0,C 180,E1 -1193.504,E2 -1193.504} C_VEL
LIN {X 0,Y 594.847,Z 280.576,A -85,B 0,C 180,E1 -1196.339,E2 -1196.339} C_VEL
LIN {X 0,Y 594.876,Z 272.807,A -85,B 0,C 180,E1 -1197.616,E2 -1197.616} C_VEL
LIN {X 0,Y 594.397,Z 270.448,A -85,B 0,C 180,E1 -1198.051,E2 -1198.051} C_VEL
LIN {X 0,Y 594.385,Z 270.448,A -85,B 0,C 180,E1 -1200.56,E2 -1200.56} C_VEL
LIN {X 0,Y 594.38,Z 270.449,A -85,B 0,C 180,E1 -1202.95,E2 -1202.95} C_VEL
LIN {X 0,Y 594.351,Z 270.454,A -85,B 0,C 180,E1 -1205.409,E2 -1205.409} C_VEL
LIN {X 0,Y 594.383,Z 270.448,A -85,B 0,C 180,E1 -1207.941,E2 -1207.941} C_VEL
LIN {X 0,Y 594.38,Z 270.449,A -85,B 0,C 180,E1 -1210.822,E2 -1210.822} C_VEL
LIN {X 0,Y 594.373,Z 270.452,A -85,B 0,C 180,E1 -1213.839,E2 -1213.839} C_VEL
LIN {X 0,Y 594.37,Z 270.45,A -85,B 0,C 180,E1 -1216.7,E2 -1216.7} C_VEL
LIN {X 0,Y 594.367,Z 270.45,A -85,B 0,C 180,E1 -1219.432,E2 -1219.432} C_VEL
LIN {X 0,Y 594.393,Z 270.449,A -85,B 0,C 180,E1 -1222.392,E2 -1222.392} C_VEL
LIN {X 0,Y 594.382,Z 270.45,A -85,B 0,C 180,E1 -1225.42,E2 -1225.42} C_VEL
LIN {X 0,Y 594.381,Z 270.449,A -85,B 0,C 180,E1 -1228.357,E2 -1228.357} C_VEL
LIN {X 0,Y 594.313,Z 270.459,A -85,B 0,C 180,E1 -1230.925,E2 -1230.925} C_VEL
LIN {X 0,Y 594.259,Z 277.195,A -85,B 0,C 180,E1 -1233.294,E2 -1233.294} C_VEL
LIN {X 0,Y 594.3,Z 283.194,A -85,B 0,C 180,E1 -1235.586,E2 -1235.586} C_VEL
LIN {X 0,Y 594.291,Z 288.519,A -85,B 0,C 180,E1 -1237.763,E2 -1237.763} C_VEL
LIN {X 0,Y 594.261,Z 295.735,A -85,B 0,C 180,E1 -1240.661,E2 -1240.661} C_VEL
LIN {X 0,Y 594.259,Z 302.951,A -85,B 0,C 180,E1 -1243.51,E2 -1243.51} C_VEL
LIN {X 0,Y 594.247,Z 310.167,A -85,B 0,C 180,E1 -1246.317,E2 -1246.317} C_VEL
LIN {X 0,Y 594.242,Z 317.383,A -85,B 0,C 180,E1 -1249.091,E2 -1249.091} C_VEL
LIN {X 0,Y 594.257,Z 324.6,A -85,B 0,C 180,E1 -1251.84,E2 -1251.84} C_VEL
LIN {X 0,Y 594.241,Z 327.701,A -85,B 0,C 180,E1 -1253.015,E2 -1253.015} C_VEL
LIN {X 0,Y 594.369,Z 337.157,A -85,B 0,C 180,E1 -1253.337,E2 -1253.337} C_VEL
LIN {X 0,Y 594.36,Z 346.41,A -85,B 0,C 180,E1 -1253.8,E2 -1253.8} C_VEL
LIN {X 0,Y 594.297,Z 355.269,A -85,B 0,C 180,E1 -1254.4,E2 -1254.4} C_VEL
LIN {X 0,Y 594.32,Z 362.742,A -85,B 0,C 180,E1 -1255.081,E2 -1255.081} C_VEL
LIN {X 0,Y 594.267,Z 368.561,A -85,B 0,C 180,E1 -1255.76,E2 -1255.76} C_VEL
LIN {X 0,Y 594.273,Z 374.023,A -85,B 0,C 180,E1 -1256.609,E2 -1256.609} C_VEL
LIN {X 0,Y 594.236,Z 377.342,A -85,B 0,C 180,E1 -1257.288,E2 -1257.288} C_VEL
LIN {X 0,Y 594.245,Z 379.827,A -85,B 0,C 180,E1 -1257.966,E2 -1257.966} C_VEL
LIN {X 0,Y 594.247,Z 381.567,A -85,B 0,C 180,E1 -1258.644,E2 -1258.644} C_VEL
LIN {X 0,Y 594.24,Z 382.615,A -85,B 0,C 180,E1 -1259.321,E2 -1259.321} C_VEL
LIN {X 0,Y 594.236,Z 382.995,A -85,B 0,C 180,E1 -1259.999,E2 -1259.999} C_VEL
LIN {X 0,Y 594.239,Z 382.714,A -85,B 0,C 180,E1 -1260.677,E2 -1260.677} C_VEL
LIN {X 0,Y 594.249,Z 381.767,A -85,B 0,C 180,E1 -1261.354,E2 -1261.354} C_VEL
LIN {X 0,Y 594.254,Z 378.996,A -85,B 0,C 180,E1 -1262.371,E2 -1262.371} C_VEL
LIN {X 0,Y 594.279,Z 376.237,A -85,B 0,C 180,E1 -1263.05,E2 -1263.05} C_VEL
LIN {X 0,Y 594.301,Z 371.552,A -85,B 0,C 180,E1 -1263.898,E2 -1263.898} C_VEL
LIN {X 0,Y 594.311,Z 366.566,A -85,B 0,C 180,E1 -1264.577,E2 -1264.577} C_VEL
LIN {X 0,Y 594.264,Z 360.259,A -85,B 0,C 180,E1 -1265.258,E2 -1265.258} C_VEL
LIN {X 0,Y 594.326,Z 353.106,A -85,B 0,C 180,E1 -1265.853,E2 -1265.853} C_VEL
LIN {X 0,Y 594.348,Z 344.427,A -85,B 0,C 180,E1 -1266.404,E2 -1266.404} C_VEL
LIN {X 0,Y 594.399,Z 335.122,A -85,B 0,C 180,E1 -1266.832,E2 -1266.832} C_VEL
LIN {X 0,Y 594.243,Z 327.662,A -85,B 0,C 180,E1 -1267.09,E2 -1267.09} C_VEL
LIN {X 0,Y 594.243,Z 321.233,A -85,B 0,C 180,E1 -1269.53,E2 -1269.53} C_VEL
LIN {X 0,Y 594.243,Z 314.014,A -85,B 0,C 180,E1 -1272.29,E2 -1272.29} C_VEL
LIN {X 0,Y 594.263,Z 307.423,A -85,B 0,C 180,E1 -1274.836,E2 -1274.836} C_VEL
LIN {X 0,Y 593.595,Z 306.053,A -85,B 0,C 180,E1 -1275.386,E2 -1275.386} C_VEL
LIN {X 0,Y 590.73,Z 303.964,A -85,B 0,C 180,E1 -1276.282,E2 -1276.282} C_VEL
LIN {X 0,Y 588.307,Z 302.315,A -85,B 0,C 180,E1 -1277.004,E2 -1277.004} C_VEL
LIN {X 0,Y 587.263,Z 300.997,A -85,B 0,C 180,E1 -1277.56,E2 -1277.56} C_VEL
LIN {X 0,Y 587.177,Z 300.533,A -85,B 0,C 180,E1 -1277.747,E2 -1277.747} C_VEL
LIN {X 0,Y 587.188,Z 294.159,A -85,B 0,C 180,E1 -1280.309,E2 -1280.309} C_VEL
LIN {X 0,Y 587.23,Z 286.927,A -85,B 0,C 180,E1 -1283.261,E2 -1283.261} C_VEL
LIN {X 0,Y 587.265,Z 279.891,A -85,B 0,C 180,E1 -1286.162,E2 -1286.162} C_VEL
LIN {X 0,Y 587.295,Z 272.427,A -85,B 0,C 180,E1 -1289.123,E2 -1289.123} C_VEL
LIN {X 0,Y 587.302,Z 271.331,A -85,B 0,C 180,E1 -1289.578,E2 -1289.578} C_VEL
LIN {X 0,Y 587.315,Z 271.322,A -85,B 0,C 180,E1 -1292.579,E2 -1292.579} C_VEL
LIN {X 0,Y 587.292,Z 271.332,A -85,B 0,C 180,E1 -1295.056,E2 -1295.056} C_VEL
LIN {X 0,Y 587.319,Z 271.321,A -85,B 0,C 180,E1 -1297.835,E2 -1297.835} C_VEL
LIN {X 0,Y 587.296,Z 271.326,A -85,B 0,C 180,E1 -1300.254,E2 -1300.254} C_VEL
LIN {X 0,Y 587.297,Z 271.327,A -85,B 0,C 180,E1 -1303.116,E2 -1303.116} C_VEL
LIN {X 0,Y 587.304,Z 271.326,A -85,B 0,C 180,E1 -1306.047,E2 -1306.047} C_VEL
LIN {X 0,Y 587.329,Z 271.322,A -85,B 0,C 180,E1 -1308.924,E2 -1308.924} C_VEL
LIN {X 0,Y 587.324,Z 271.322,A -85,B 0,C 180,E1 -1311.52,E2 -1311.52} C_VEL
LIN {X 0,Y 587.342,Z 271.322,A -85,B 0,C 180,E1 -1314.454,E2 -1314.454} C_VEL
LIN {X 0,Y 587.332,Z 271.32,A -85,B 0,C 180,E1 -1316.887,E2 -1316.887} C_VEL
LIN {X 0,Y 587.342,Z 271.324,A -85,B 0,C 180,E1 -1319.487,E2 -1319.487} C_VEL
LIN {X 0,Y 587.342,Z 271.319,A -85,B 0,C 180,E1 -1322.306,E2 -1322.306} C_VEL
LIN {X 0,Y 587.329,Z 271.32,A -85,B 0,C 180,E1 -1324.483,E2 -1324.483} C_VEL
LIN {X 0,Y 587.331,Z 271.326,A -85,B 0,C 180,E1 -1327.486,E2 -1327.486} C_VEL
LIN {X 0,Y 587.321,Z 271.323,A -85,B 0,C 180,E1 -1329.695,E2 -1329.695} C_VEL
LIN {X 0,Y 587.347,Z 271.321,A -85,B 0,C 180,E1 -1332.594,E2 -1332.594} C_VEL
LIN {X 0,Y 587.353,Z 271.317,A -85,B 0,C 180,E1 -1335.739,E2 -1335.739} C_VEL
LIN {X 0,Y 587.335,Z 271.325,A -85,B 0,C 180,E1 -1338.866,E2 -1338.866} C_VEL
LIN {X 0,Y 587.347,Z 271.318,A -85,B 0,C 180,E1 -1341.744,E2 -1341.744} C_VEL
LIN {X 0,Y 587.338,Z 271.325,A -85,B 0,C 180,E1 -1344.507,E2 -1344.507} C_VEL
LIN {X 0,Y 587.326,Z 271.32,A -85,B 0,C 180,E1 -1347.257,E2 -1347.257} C_VEL
LIN {X 0,Y 587.369,Z 271.324,A -85,B 0,C 180,E1 -1350,E2 -1350} C_VEL
LIN {X 0,Y 587.328,Z 271.32,A -85,B 0,C 180,E1 -1352.743,E2 -1352.743} C_VEL
LIN {X 0,Y 587.34,Z 271.325,A -85,B 0,C 180,E1 -1355.493,E2 -1355.493} C_VEL
LIN {X 0,Y 587.348,Z 271.318,A -85,B 0,C 180,E1 -1358.256,E2 -1358.256} C_VEL
LIN {X 0,Y 587.335,Z 271.325,A -85,B 0,C 180,E1 -1361.134,E2 -1361.134} C_VEL
LIN {X 0,Y 587.353,Z 271.317,A -85,B 0,C 180,E1 -1364.261,E2 -1364.261} C_VEL
LIN {X 0,Y 587.346,Z 271.321,A -85,B 0,C 180,E1 -1367.406,E2 -1367.406} C_VEL
LIN {X 0,Y 587.322,Z 271.323,A -85,B 0,C 180,E1 -1370.305,E2 -1370.305} C_VEL
LIN {X 0,Y 587.314,Z 271.323,A -85,B 0,C 180,E1 -1373.259,E2 -1373.259} C_VEL
LIN {X 0,Y 587.33,Z 271.32,A -85,B 0,C 180,E1 -1375.517,E2 -1375.517} C_VEL
LIN {X 0,Y 587.34,Z 271.321,A -85,B 0,C 180,E1 -1377.818,E2 -1377.818} C_VEL
LIN {X 0,Y 587.342,Z 271.324,A -85,B 0,C 180,E1 -1380.513,E2 -1380.513} C_VEL
LIN {X 0,Y 587.329,Z 271.321,A -85,B 0,C 180,E1 -1383.397,E2 -1383.397} C_VEL
LIN {X 0,Y 587.347,Z 271.327,A -85,B 0,C 180,E1 -1385.896,E2 -1385.896} C_VEL
LIN {X 0,Y 587.324,Z 271.321,A -85,B 0,C 180,E1 -1388.48,E2 -1388.48} C_VEL
LIN {X 0,Y 587.329,Z 271.323,A -85,B 0,C 180,E1 -1391.158,E2 -1391.158} C_VEL
LIN {X 0,Y 587.304,Z 271.324,A -85,B 0,C 180,E1 -1394.113,E2 -1394.113} C_VEL
LIN {X 0,Y 587.298,Z 271.329,A -85,B 0,C 180,E1 -1396.994,E2 -1396.994} C_VEL
LIN {X 0,Y 587.296,Z 271.325,A -85,B 0,C 180,E1 -1399.746,E2 -1399.746} C_VEL
LIN {X 0,Y 587.331,Z 271.321,A -85,B 0,C 180,E1 -1402.393,E2 -1402.393} C_VEL
LIN {X 0,Y 587.315,Z 271.322,A -85,B 0,C 180,E1 -1405.657,E2 -1405.657} C_VEL
LIN {X 0,Y 587.327,Z 271.323,A -85,B 0,C 180,E1 -1408.232,E2 -1408.232} C_VEL
LIN {X 0,Y 587.324,Z 271.344,A -85,B 0,C 180,E1 -1410.226,E2 -1410.226} C_VEL
LIN {X 0,Y 587.299,Z 277.836,A -85,B 0,C 180,E1 -1412.954,E2 -1412.954} C_VEL
LIN {X 0,Y 587.25,Z 283.663,A -85,B 0,C 180,E1 -1415.443,E2 -1415.443} C_VEL
LIN {X 0,Y 587.205,Z 290.33,A -85,B 0,C 180,E1 -1418.222,E2 -1418.222} C_VEL
LIN {X 0,Y 587.221,Z 297.545,A -85,B 0,C 180,E1 -1421.148,E2 -1421.148} C_VEL
LIN {X 0,Y 587.171,Z 304.761,A -85,B 0,C 180,E1 -1424.022,E2 -1424.022} C_VEL
LIN {X 0,Y 587.183,Z 310.173,A -85,B 0,C 180,E1 -1426.151,E2 -1426.151} C_VEL
LIN {X 0,Y 587.165,Z 317.39,A -85,B 0,C 180,E1 -1428.96,E2 -1428.96} C_VEL
LIN {X 0,Y 587.158,Z 324.606,A -85,B 0,C 180,E1 -1431.743,E2 -1431.743} C_VEL
LIN {X 0,Y 587.154,Z 327.741,A -85,B 0,C 180,E1 -1432.932,E2 -1432.932} C_VEL
LIN {X 0,Y 587.333,Z 336.939,A -85,B 0,C 180,E1 -1433.25,E2 -1433.25} C_VEL
LIN {X 0,Y 587.313,Z 344.782,A -85,B 0,C 180,E1 -1433.633,E2 -1433.633} C_VEL
LIN {X 0,Y 587.274,Z 351.819,A -85,B 0,C 180,E1 -1434.077,E2 -1434.077} C_VEL
LIN {X 0,Y 587.178,Z 359.268,A -85,B 0,C 180,E1 -1434.679,E2 -1434.679} C_VEL
LIN {X 0,Y 587.245,Z 365.807,A -85,B 0,C 180,E1 -1435.367,E2 -1435.367} C_VEL
LIN {X 0,Y 587.223,Z 370.93,A -85,B 0,C 180,E1 -1436.055,E2 -1436.055} C_VEL
LIN {X 0,Y 587.183,Z 375.832,A -85,B 0,C 180,E1 -1436.913,E2 -1436.913} C_VEL
LIN {X 0,Y 587.147,Z 379.846,A -85,B 0,C 180,E1 -1437.943,E2 -1437.943} C_VEL
LIN {X 0,Y 587.147,Z 381.571,A -85,B 0,C 180,E1 -1438.629,E2 -1438.629} C_VEL
LIN {X 0,Y 587.14,Z 382.597,A -85,B 0,C 180,E1 -1439.315,E2 -1439.315} C_VEL
LIN {X 0,Y 587.137,Z 382.972,A -85,B 0,C 180,E1 -1440.001,E2 -1440.001} C_VEL
LIN {X 0,Y 587.14,Z 382.701,A -85,B 0,C 180,E1 -1440.687,E2 -1440.687} C_VEL
LIN {X 0,Y 587.149,Z 381.762,A -85,B 0,C 180,E1 -1441.373,E2 -1441.373} C_VEL
LIN {X 0,Y 587.172,Z 378.996,A -85,B 0,C 180,E1 -1442.402,E2 -1442.402} C_VEL
LIN {X 0,Y 587.184,Z 376.239,A -85,B 0,C 180,E1 -1443.088,E2 -1443.088} C_VEL
LIN {X 0,Y 587.223,Z 371.521,A -85,B 0,C 180,E1 -1443.947,E2 -1443.947} C_VEL
LIN {X 0,Y 587.247,Z 366.537,A -85,B 0,C 180,E1 -1444.634,E2 -1444.634} C_VEL
LIN {X 0,Y 587.183,Z 360.216,A -85,B 0,C 180,E1 -1445.323,E2 -1445.323} C_VEL
LIN {X 0,Y 587.274,Z 353.041,A -85,B 0,C 180,E1 -1445.925,E2 -1445.925} C_VEL
LIN {X 0,Y 587.3,Z 345.356,A -85,B 0,C 180,E1 -1446.425,E2 -1446.425} C_VEL
LIN {X 0,Y 587.313,Z 337.602,A -85,B 0,C 180,E1 -1446.812,E2 -1446.812} C_VEL
LIN {X 0,Y 587.232,Z 328.588,A -85,B 0,C 180,E1 -1447.134,E2 -1447.134} C_VEL
LIN {X 0,Y 587.158,Z 327.656,A -85,B 0,C 180,E1 -1447.178,E2 -1447.178} C_VEL
LIN {X 0,Y 587.143,Z 321.227,A -85,B 0,C 180,E1 -1449.648,E2 -1449.648} C_VEL
LIN {X 0,Y 587.164,Z 314.008,A -85,B 0,C 180,E1 -1452.443,E2 -1452.443} C_VEL
LIN {X 0,Y 587.204,Z 308.594,A -85,B 0,C 180,E1 -1454.558,E2 -1454.558} C_VEL
LIN {X 0,Y 587.199,Z 301.374,A -85,B 0,C 180,E1 -1457.411,E2 -1457.411} C_VEL
LIN {X 0,Y 587.207,Z 295.96,A -85,B 0,C 180,E1 -1459.58,E2 -1459.58} C_VEL
LIN {X 0,Y 587.242,Z 288.74,A -85,B 0,C 180,E1 -1462.518,E2 -1462.518} C_VEL
LIN {X 0,Y 587.317,Z 281.929,A -85,B 0,C 180,E1 -1465.518,E2 -1465.518} C_VEL
LIN {X 0,Y 587.301,Z 276.209,A -85,B 0,C 180,E1 -1467.821,E2 -1467.821} C_VEL
LIN {X 0,Y 587.333,Z 271.327,A -85,B 0,C 180,E1 -1469.874,E2 -1469.874} C_VEL
LIN {X 0,Y 587.342,Z 271.327,A -85,B 0,C 180,E1 -1472.579,E2 -1472.579} C_VEL
LIN {X 0,Y 587.334,Z 271.327,A -85,B 0,C 180,E1 -1475.056,E2 -1475.056} C_VEL
LIN {X 0,Y 587.344,Z 271.327,A -85,B 0,C 180,E1 -1477.839,E2 -1477.839} C_VEL
LIN {X 0,Y 587.317,Z 271.329,A -85,B 0,C 180,E1 -1480.255,E2 -1480.255} C_VEL
LIN {X 0,Y 587.321,Z 271.33,A -85,B 0,C 180,E1 -1483.118,E2 -1483.118} C_VEL
LIN {X 0,Y 587.317,Z 271.328,A -85,B 0,C 180,E1 -1486.049,E2 -1486.049} C_VEL
LIN {X 0,Y 587.341,Z 271.325,A -85,B 0,C 180,E1 -1488.925,E2 -1488.925} C_VEL
LIN {X 0,Y 587.327,Z 271.329,A -85,B 0,C 180,E1 -1491.52,E2 -1491.52} C_VEL
LIN {X 0,Y 587.294,Z 271.331,A -85,B 0,C 180,E1 -1494.1,E2 -1494.1} C_VEL
LIN {X 0,Y 587.337,Z 271.327,A -85,B 0,C 180,E1 -1496.603,E2 -1496.603} C_VEL
LIN {X 0,Y 587.341,Z 271.326,A -85,B 0,C 180,E1 -1499.49,E2 -1499.49} C_VEL
LIN {X 0,Y 587.369,Z 271.435,A -85,B 0,C 180,E1 -1501.722,E2 -1501.722} C_VEL
LIN {X 0,Y 588.057,Z 274.746,A -85,B 0,C 180,E1 -1502.329,E2 -1502.329} C_VEL
LIN {X 0,Y 587.88,Z 290.053,A -85,B 0,C 180,E1 -1504.887,E2 -1504.887} C_VEL
LIN {X 0,Y 587.734,Z 307.361,A -85,B 0,C 180,E1 -1507.687,E2 -1507.687} C_VEL
LIN {X 0,Y 587.615,Z 326.501,A -85,B 0,C 180,E1 -1510.723,E2 -1510.723} C_VEL
LIN {X 0,Y 587.479,Z 345.44,A -85,B 0,C 180,E1 -1513.672,E2 -1513.672} C_VEL
LIN {X 0,Y 587.381,Z 363.903,A -85,B 0,C 180,E1 -1516.508,E2 -1516.508} C_VEL
LIN {X 0,Y 587.361,Z 372.199,A -85,B 0,C 180,E1 -1517.749,E2 -1517.749} C_VEL
LIN {X 0,Y 587.724,Z 377.607,A -85,B 0,C 180,E1 -1517.833,E2 -1517.833} C_VEL
LIN {X 0,Y 587.688,Z 390.69,A -85,B 0,C 180,E1 -1518.117,E2 -1518.117} C_VEL
LIN {X 0,Y 587.615,Z 403.934,A -85,B 0,C 180,E1 -1518.558,E2 -1518.558} C_VEL
LIN {X 0,Y 587.547,Z 416.631,A -85,B 0,C 180,E1 -1519.141,E2 -1519.141} C_VEL
LIN {X 0,Y 587.468,Z 428.201,A -85,B 0,C 180,E1 -1519.836,E2 -1519.836} C_VEL
LIN {X 0,Y 587.367,Z 438.597,A -85,B 0,C 180,E1 -1520.617,E2 -1520.617} C_VEL
LIN {X 0,Y 587.322,Z 447.112,A -85,B 0,C 180,E1 -1521.398,E2 -1521.398} C_VEL
LIN {X 0,Y 587.274,Z 454.96,A -85,B 0,C 180,E1 -1522.263,E2 -1522.263} C_VEL
LIN {X 0,Y 587.231,Z 461.469,A -85,B 0,C 180,E1 -1523.126,E2 -1523.126} C_VEL
LIN {X 0,Y 587.237,Z 467.866,A -85,B 0,C 180,E1 -1524.161,E2 -1524.161} C_VEL
LIN {X 0,Y 587.147,Z 472.949,A -85,B 0,C 180,E1 -1525.194,E2 -1525.194} C_VEL
LIN {X 0,Y 587.213,Z 476.896,A -85,B 0,C 180,E1 -1526.226,E2 -1526.226} C_VEL
LIN {X 0,Y 587.132,Z 479.81,A -85,B 0,C 180,E1 -1527.256,E2 -1527.256} C_VEL
LIN {X 0,Y 587.141,Z 481.201,A -85,B 0,C 180,E1 -1527.942,E2 -1527.942} C_VEL
LIN {X 0,Y 587.14,Z 482.784,A -85,B 0,C 180,E1 -1529.314,E2 -1529.314} C_VEL
LIN {X 0,Y 587.137,Z 483,A -85,B 0,C 180,E1 -1530,E2 -1530} C_VEL
LIN {X 0,Y 587.147,Z 482.185,A -85,B 0,C 180,E1 -1531.372,E2 -1531.372} C_VEL
LIN {X 0,Y 587.141,Z 481.2,A -85,B 0,C 180,E1 -1532.058,E2 -1532.058} C_VEL
LIN {X 0,Y 587.132,Z 479.808,A -85,B 0,C 180,E1 -1532.744,E2 -1532.744} C_VEL
LIN {X 0,Y 587.213,Z 476.896,A -85,B 0,C 180,E1 -1533.774,E2 -1533.774} C_VEL
LIN {X 0,Y 587.147,Z 472.95,A -85,B 0,C 180,E1 -1534.806,E2 -1534.806} C_VEL
LIN {X 0,Y 587.218,Z 466.877,A -85,B 0,C 180,E1 -1536.011,E2 -1536.011} C_VEL
LIN {X 0,Y 587.245,Z 460.237,A -85,B 0,C 180,E1 -1537.046,E2 -1537.046} C_VEL
LIN {X 0,Y 587.3,Z 451.99,A -85,B 0,C 180,E1 -1538.083,E2 -1538.083} C_VEL
LIN {X 0,Y 587.343,Z 443.537,A -85,B 0,C 180,E1 -1538.949,E2 -1538.949} C_VEL
LIN {X 0,Y 587.42,Z 433.094,A -85,B 0,C 180,E1 -1539.816,E2 -1539.816} C_VEL
LIN {X 0,Y 587.508,Z 422.756,A -85,B 0,C 180,E1 -1540.511,E2 -1540.511} C_VEL
LIN {X 0,Y 587.567,Z 411,A -85,B 0,C 180,E1 -1541.14,E2 -1541.14} C_VEL
LIN {X 0,Y 587.617,Z 398.61,A -85,B 0,C 180,E1 -1541.639,E2 -1541.639} C_VEL
LIN {X 0,Y 587.677,Z 385.436,A -85,B 0,C 180,E1 -1542.015,E2 -1542.015} C_VEL
LIN {X 0,Y 587.515,Z 373.279,A -85,B 0,C 180,E1 -1542.234,E2 -1542.234} C_VEL
LIN {X 0,Y 587.345,Z 371.981,A -85,B 0,C 180,E1 -1542.263,E2 -1542.263} C_VEL
LIN {X 0,Y 587.454,Z 353.518,A -85,B 0,C 180,E1 -1545.082,E2 -1545.082} C_VEL
LIN {X 0,Y 587.527,Z 335.055,A -85,B 0,C 180,E1 -1547.94,E2 -1547.94} C_VEL
LIN {X 0,Y 587.658,Z 317.747,A -85,B 0,C 180,E1 -1550.659,E2 -1550.659} C_VEL
LIN {X 0,Y 587.84,Z 299.284,A -85,B 0,C 180,E1 -1553.61,E2 -1553.61} C_VEL
LIN {X 0,Y 587.996,Z 280.821,A -85,B 0,C 180,E1 -1556.629,E2 -1556.629} C_VEL
LIN {X 0,Y 587.882,Z 273.875,A -85,B 0,C 180,E1 -1557.79,E2 -1557.79} C_VEL
LIN {X 0,Y 587.359,Z 271.324,A -85,B 0,C 180,E1 -1558.254,E2 -1558.254} C_VEL
LIN {X 0,Y 587.333,Z 271.328,A -85,B 0,C 180,E1 -1560.967,E2 -1560.967} C_VEL
LIN {X 0,Y 587.331,Z 271.328,A -85,B 0,C 180,E1 -1563.397,E2 -1563.397} C_VEL
LIN {X 0,Y 587.294,Z 271.331,A -85,B 0,C 180,E1 -1565.9,E2 -1565.9} C_VEL
LIN {X 0,Y 587.328,Z 271.329,A -85,B 0,C 180,E1 -1568.48,E2 -1568.48} C_VEL
LIN {X 0,Y 587.34,Z 271.325,A -85,B 0,C 180,E1 -1571.157,E2 -1571.157} C_VEL
LIN {X 0,Y 587.332,Z 271.327,A -85,B 0,C 180,E1 -1574.113,E2 -1574.113} C_VEL
LIN {X 0,Y 587.317,Z 271.331,A -85,B 0,C 180,E1 -1576.993,E2 -1576.993} C_VEL
LIN {X 0,Y 587.32,Z 271.327,A -85,B 0,C 180,E1 -1579.745,E2 -1579.745} C_VEL
LIN {X 0,Y 587.349,Z 271.326,A -85,B 0,C 180,E1 -1582.392,E2 -1582.392} C_VEL
LIN {X 0,Y 587.346,Z 271.326,A -85,B 0,C 180,E1 -1585.653,E2 -1585.653} C_VEL
LIN {X 0,Y 587.346,Z 271.325,A -85,B 0,C 180,E1 -1588.231,E2 -1588.231} C_VEL
LIN {X 0,Y 587.279,Z 271.336,A -85,B 0,C 180,E1 -1590.948,E2 -1590.948} C_VEL
LIN {X 0,Y 587.229,Z 271.491,A -85,B 0,C 180,E1 -1591.137,E2 -1591.137} C_VEL
LIN {X 0,Y 587.199,Z 276.786,A -85,B 0,C 180,E1 -1592.947,E2 -1592.947} C_VEL
LIN {X 0,Y 587.199,Z 283.445,A -85,B 0,C 180,E1 -1595.453,E2 -1595.453} C_VEL
LIN {X 0,Y 587.241,Z 288.521,A -85,B 0,C 180,E1 -1597.482,E2 -1597.482} C_VEL
LIN {X 0,Y 587.193,Z 295.736,A -85,B 0,C 180,E1 -1600.419,E2 -1600.419} C_VEL
LIN {X 0,Y 587.17,Z 302.952,A -85,B 0,C 180,E1 -1603.305,E2 -1603.305} C_VEL
LIN {X 0,Y 587.186,Z 310.168,A -85,B 0,C 180,E1 -1606.149,E2 -1606.149} C_VEL
LIN {X 0,Y 587.168,Z 317.385,A -85,B 0,C 180,E1 -1608.958,E2 -1608.958} C_VEL
LIN {X 0,Y 587.16,Z 324.602,A -85,B 0,C 180,E1 -1611.741,E2 -1611.741} C_VEL
LIN {X 0,Y 587.155,Z 327.703,A -85,B 0,C 180,E1 -1612.93,E2 -1612.93} C_VEL
LIN {X 0,Y 587.326,Z 336.677,A -85,B 0,C 180,E1 -1613.238,E2 -1613.238} C_VEL
LIN {X 0,Y 587.312,Z 345.886,A -85,B 0,C 180,E1 -1613.694,E2 -1613.694} C_VEL
LIN {X 0,Y 587.245,Z 354.173,A -85,B 0,C 180,E1 -1614.247,E2 -1614.247} C_VEL
LIN {X 0,Y 587.237,Z 361.055,A -85,B 0,C 180,E1 -1614.849,E2 -1614.849} C_VEL
LIN {X 0,Y 587.216,Z 367.221,A -85,B 0,C 180,E1 -1615.537,E2 -1615.537} C_VEL
LIN {X 0,Y 587.228,Z 372.065,A -85,B 0,C 180,E1 -1616.225,E2 -1616.225} C_VEL
LIN {X 0,Y 587.183,Z 375.83,A -85,B 0,C 180,E1 -1616.912,E2 -1616.912} C_VEL
LIN {X 0,Y 587.146,Z 379.827,A -85,B 0,C 180,E1 -1617.941,E2 -1617.941} C_VEL
LIN {X 0,Y 587.147,Z 381.568,A -85,B 0,C 180,E1 -1618.627,E2 -1618.627} C_VEL
LIN {X 0,Y 587.14,Z 382.615,A -85,B 0,C 180,E1 -1619.313,E2 -1619.313} C_VEL
LIN {X 0,Y 587.137,Z 382.996,A -85,B 0,C 180,E1 -1619.999,E2 -1619.999} C_VEL
LIN {X 0,Y 587.14,Z 382.714,A -85,B 0,C 180,E1 -1620.685,E2 -1620.685} C_VEL
LIN {X 0,Y 587.148,Z 381.766,A -85,B 0,C 180,E1 -1621.371,E2 -1621.371} C_VEL
LIN {X 0,Y 587.172,Z 378.996,A -85,B 0,C 180,E1 -1622.4,E2 -1622.4} C_VEL
LIN {X 0,Y 587.184,Z 376.238,A -85,B 0,C 180,E1 -1623.087,E2 -1623.087} C_VEL
LIN {X 0,Y 587.223,Z 371.544,A -85,B 0,C 180,E1 -1623.945,E2 -1623.945} C_VEL
LIN {X 0,Y 587.258,Z 365.145,A -85,B 0,C 180,E1 -1624.804,E2 -1624.804} C_VEL
LIN {X 0,Y 587.204,Z 358.371,A -85,B 0,C 180,E1 -1625.493,E2 -1625.493} C_VEL
LIN {X 0,Y 587.293,Z 350.674,A -85,B 0,C 180,E1 -1626.096,E2 -1626.096} C_VEL
LIN {X 0,Y 587.304,Z 341.565,A -85,B 0,C 180,E1 -1626.63,E2 -1626.63} C_VEL
LIN {X 0,Y 587.369,Z 332.719,A -85,B 0,C 180,E1 -1627.001,E2 -1627.001} C_VEL
LIN {X 0,Y 587.158,Z 327.66,A -85,B 0,C 180,E1 -1627.176,E2 -1627.176} C_VEL
LIN {X 0,Y 587.155,Z 321.231,A -85,B 0,C 180,E1 -1629.646,E2 -1629.646} C_VEL
LIN {X 0,Y 587.16,Z 314.013,A -85,B 0,C 180,E1 -1632.441,E2 -1632.441} C_VEL
LIN {X 0,Y 587.177,Z 307.87,A -85,B 0,C 180,E1 -1634.842,E2 -1634.842} C_VEL
LIN {X 0,Y 587.177,Z 300.533,A -85,B 0,C 180,E1 -1637.747,E2 -1637.747} C_VEL
LIN {X 0,Y 586.507,Z 299.192,A -85,B 0,C 180,E1 -1638.305,E2 -1638.305} C_VEL
LIN {X 0,Y 583.658,Z 297.172,A -85,B 0,C 180,E1 -1639.213,E2 -1639.213} C_VEL
LIN {X 0,Y 581.256,Z 295.58,A -85,B 0,C 180,E1 -1639.944,E2 -1639.944} C_VEL
LIN {X 0,Y 580.225,Z 294.296,A -85,B 0,C 180,E1 -1640.507,E2 -1640.507} C_VEL
LIN {X 0,Y 580.142,Z 293.842,A -85,B 0,C 180,E1 -1640.697,E2 -1640.697} C_VEL
LIN {X 0,Y 580.171,Z 288.362,A -85,B 0,C 180,E1 -1642.98,E2 -1642.98} C_VEL
LIN {X 0,Y 580.191,Z 281.374,A -85,B 0,C 180,E1 -1645.853,E2 -1645.853} C_VEL
LIN {X 0,Y 580.239,Z 273.54,A -85,B 0,C 180,E1 -1648.978,E2 -1648.978} C_VEL
LIN {X 0,Y 580.244,Z 272.211,A -85,B 0,C 180,E1 -1649.504,E2 -1649.504} C_VEL
LIN {X 0,Y 580.276,Z 272.198,A -85,B 0,C 180,E1 -1652.2,E2 -1652.2} C_VEL
LIN {X 0,Y 580.266,Z 272.202,A -85,B 0,C 180,E1 -1654.696,E2 -1654.696} C_VEL
LIN {X 0,Y 580.279,Z 272.204,A -85,B 0,C 180,E1 -1657.268,E2 -1657.268} C_VEL
LIN {X 0,Y 580.276,Z 272.2,A -85,B 0,C 180,E1 -1660.268,E2 -1660.268} C_VEL
LIN {X 0,Y 580.265,Z 272.209,A -85,B 0,C 180,E1 -1662.706,E2 -1662.706} C_VEL
LIN {X 0,Y 580.25,Z 272.202,A -85,B 0,C 180,E1 -1665.609,E2 -1665.609} C_VEL
LIN {X 0,Y 580.271,Z 272.206,A -85,B 0,C 180,E1 -1668.23,E2 -1668.23} C_VEL
LIN {X 0,Y 580.284,Z 272.198,A -85,B 0,C 180,E1 -1670.965,E2 -1670.965} C_VEL
LIN {X 0,Y 580.288,Z 272.2,A -85,B 0,C 180,E1 -1673.598,E2 -1673.598} C_VEL
LIN {X 0,Y 580.312,Z 272.2,A -85,B 0,C 180,E1 -1676.145,E2 -1676.145} C_VEL
LIN {X 0,Y 580.282,Z 272.198,A -85,B 0,C 180,E1 -1678.615,E2 -1678.615} C_VEL
LIN {X 0,Y 580.289,Z 272.199,A -85,B 0,C 180,E1 -1681.024,E2 -1681.024} C_VEL
LIN {X 0,Y 580.319,Z 272.201,A -85,B 0,C 180,E1 -1683.658,E2 -1683.658} C_VEL
LIN {X 0,Y 580.27,Z 272.2,A -85,B 0,C 180,E1 -1686.442,E2 -1686.442} C_VEL
LIN {X 0,Y 580.271,Z 272.205,A -85,B 0,C 180,E1 -1689.437,E2 -1689.437} C_VEL
LIN {X 0,Y 580.268,Z 272.201,A -85,B 0,C 180,E1 -1691.645,E2 -1691.645} C_VEL
LIN {X 0,Y 580.266,Z 272.2,A -85,B 0,C 180,E1 -1693.825,E2 -1693.825} C_VEL
LIN {X 0,Y 580.316,Z 272.194,A -85,B 0,C 180,E1 -1695.983,E2 -1695.983} C_VEL
LIN {X 0,Y 580.292,Z 272.203,A -85,B 0,C 180,E1 -1698.827,E2 -1698.827} C_VEL
LIN {X 0,Y 580.31,Z 272.195,A -85,B 0,C 180,E1 -1701.644,E2 -1701.644} C_VEL
LIN {X 0,Y 580.306,Z 272.202,A -85,B 0,C 180,E1 -1704.44,E2 -1704.44} C_VEL
LIN {X 0,Y 580.333,Z 272.198,A -85,B 0,C 180,E1 -1707.918,E2 -1707.918} C_VEL
LIN {X 0,Y 580.337,Z 272.2,A -85,B 0,C 180,E1 -1710,E2 -1710} C_VEL
LIN {X 0,Y 580.296,Z 272.196,A -85,B 0,C 180,E1 -1712.777,E2 -1712.777} C_VEL
LIN {X 0,Y 580.308,Z 272.202,A -85,B 0,C 180,E1 -1715.56,E2 -1715.56} C_VEL
LIN {X 0,Y 580.311,Z 272.194,A -85,B 0,C 180,E1 -1718.356,E2 -1718.356} C_VEL
LIN {X 0,Y 580.287,Z 272.204,A -85,B 0,C 180,E1 -1721.191,E2 -1721.191} C_VEL
LIN {X 0,Y 580.316,Z 272.194,A -85,B 0,C 180,E1 -1724.017,E2 -1724.017} C_VEL
LIN {X 0,Y 580.3,Z 272.204,A -85,B 0,C 180,E1 -1726.914,E2 -1726.914} C_VEL
LIN {X 0,Y 580.296,Z 272.196,A -85,B 0,C 180,E1 -1729.823,E2 -1729.823} C_VEL
LIN {X 0,Y 580.266,Z 272.201,A -85,B 0,C 180,E1 -1732.053,E2 -1732.053} C_VEL
LIN {X 0,Y 580.299,Z 272.198,A -85,B 0,C 180,E1 -1735.08,E2 -1735.08} C_VEL
LIN {X 0,Y 580.311,Z 272.197,A -85,B 0,C 180,E1 -1737.864,E2 -1737.864} C_VEL
LIN {X 0,Y 580.291,Z 272.2,A -85,B 0,C 180,E1 -1740.698,E2 -1740.698} C_VEL
LIN {X 0,Y 580.297,Z 272.197,A -85,B 0,C 180,E1 -1743.318,E2 -1743.318} C_VEL
LIN {X 0,Y 580.317,Z 272.201,A -85,B 0,C 180,E1 -1745.768,E2 -1745.768} C_VEL
LIN {X 0,Y 580.28,Z 272.202,A -85,B 0,C 180,E1 -1748.147,E2 -1748.147} C_VEL
LIN {X 0,Y 580.292,Z 272.197,A -85,B 0,C 180,E1 -1750.844,E2 -1750.844} C_VEL
LIN {X 0,Y 580.265,Z 272.207,A -85,B 0,C 180,E1 -1753.659,E2 -1753.659} C_VEL
LIN {X 0,Y 580.236,Z 272.204,A -85,B 0,C 180,E1 -1756.614,E2 -1756.614} C_VEL
LIN {X 0,Y 580.287,Z 272.206,A -85,B 0,C 180,E1 -1759.157,E2 -1759.157} C_VEL
LIN {X 0,Y 580.276,Z 272.198,A -85,B 0,C 180,E1 -1761.929,E2 -1761.929} C_VEL
LIN {X 0,Y 580.215,Z 272.209,A -85,B 0,C 180,E1 -1764.452,E2 -1764.452} C_VEL
LIN {X 0,Y 580.274,Z 272.204,A -85,B 0,C 180,E1 -1766.976,E2 -1766.976} C_VEL
LIN {X 0,Y 580.297,Z 272.2,A -85,B 0,C 180,E1 -1770.129,E2 -1770.129} C_VEL
LIN {X 0,Y 580.259,Z 276.756,A -85,B 0,C 180,E1 -1772.149,E2 -1772.149} C_VEL
LIN {X 0,Y 580.226,Z 283.343,A -85,B 0,C 180,E1 -1774.918,E2 -1774.918} C_VEL
LIN {X 0,Y 580.163,Z 290.333,A -85,B 0,C 180,E1 -1777.944,E2 -1777.944} C_VEL
LIN {X 0,Y 580.137,Z 297.547,A -85,B 0,C 180,E1 -1780.909,E2 -1780.909} C_VEL
LIN {X 0,Y 580.094,Z 304.762,A -85,B 0,C 180,E1 -1783.821,E2 -1783.821} C_VEL
LIN {X 0,Y 580.13,Z 310.175,A -85,B 0,C 180,E1 -1785.979,E2 -1785.979} C_VEL
LIN {X 0,Y 580.098,Z 317.617,A -85,B 0,C 180,E1 -1788.913,E2 -1788.913} C_VEL
LIN {X 0,Y 580.075,Z 324.608,A -85,B 0,C 180,E1 -1791.641,E2 -1791.641} C_VEL
LIN {X 0,Y 580.066,Z 327.771,A -85,B 0,C 180,E1 -1792.845,E2 -1792.845} C_VEL
LIN {X 0,Y 580.308,Z 335.703,A -85,B 0,C 180,E1 -1793.115,E2 -1793.115} C_VEL
LIN {X 0,Y 580.253,Z 344.747,A -85,B 0,C 180,E1 -1793.553,E2 -1793.553} C_VEL
LIN {X 0,Y 580.222,Z 351.829,A -85,B 0,C 180,E1 -1794.004,E2 -1794.004} C_VEL
LIN {X 0,Y 580.104,Z 359.261,A -85,B 0,C 180,E1 -1794.613,E2 -1794.613} C_VEL
LIN {X 0,Y 580.179,Z 365.81,A -85,B 0,C 180,E1 -1795.311,E2 -1795.311} C_VEL
LIN {X 0,Y 580.133,Z 370.927,A -85,B 0,C 180,E1 -1796.007,E2 -1796.007} C_VEL
LIN {X 0,Y 580.095,Z 375.83,A -85,B 0,C 180,E1 -1796.876,E2 -1796.876} C_VEL
LIN {X 0,Y 580.049,Z 379.852,A -85,B 0,C 180,E1 -1797.918,E2 -1797.918} C_VEL
LIN {X 0,Y 580.047,Z 381.571,A -85,B 0,C 180,E1 -1798.612,E2 -1798.612} C_VEL
LIN {X 0,Y 580.041,Z 382.591,A -85,B 0,C 180,E1 -1799.307,E2 -1799.307} C_VEL
LIN {X 0,Y 580.038,Z 382.963,A -85,B 0,C 180,E1 -1800.001,E2 -1800.001} C_VEL
LIN {X 0,Y 580.04,Z 382.695,A -85,B 0,C 180,E1 -1800.695,E2 -1800.695} C_VEL
LIN {X 0,Y 580.048,Z 381.761,A -85,B 0,C 180,E1 -1801.389,E2 -1801.389} C_VEL
LIN {X 0,Y 580.093,Z 378.998,A -85,B 0,C 180,E1 -1802.431,E2 -1802.431} C_VEL
LIN {X 0,Y 580.095,Z 376.242,A -85,B 0,C 180,E1 -1803.126,E2 -1803.126} C_VEL
LIN {X 0,Y 580.133,Z 371.51,A -85,B 0,C 180,E1 -1803.995,E2 -1803.995} C_VEL
LIN {X 0,Y 580.182,Z 366.533,A -85,B 0,C 180,E1 -1804.691,E2 -1804.691} C_VEL
LIN {X 0,Y 580.108,Z 360.197,A -85,B 0,C 180,E1 -1805.388,E2 -1805.388} C_VEL
LIN {X 0,Y 580.221,Z 353.022,A -85,B 0,C 180,E1 -1805.998,E2 -1805.998} C_VEL
LIN {X 0,Y 580.229,Z 345.337,A -85,B 0,C 180,E1 -1806.503,E2 -1806.503} C_VEL
LIN {X 0,Y 580.276,Z 337.766,A -85,B 0,C 180,E1 -1806.886,E2 -1806.886} C_VEL
LIN {X 0,Y 580.175,Z 328.901,A -85,B 0,C 180,E1 -1807.21,E2 -1807.21} C_VEL
LIN {X 0,Y 580.055,Z 327.654,A -85,B 0,C 180,E1 -1807.266,E2 -1807.266} C_VEL
LIN {X 0,Y 580.052,Z 321.225,A -85,B 0,C 180,E1 -1809.767,E2 -1809.767} C_VEL
LIN {X 0,Y 580.088,Z 315.811,A -85,B 0,C 180,E1 -1811.887,E2 -1811.887} C_VEL
LIN {X 0,Y 580.12,Z 308.592,A -85,B 0,C 180,E1 -1814.739,E2 -1814.739} C_VEL
LIN {X 0,Y 580.13,Z 301.373,A -85,B 0,C 180,E1 -1817.63,E2 -1817.63} C_VEL
LIN {X 0,Y 580.129,Z 295.958,A -85,B 0,C 180,E1 -1819.829,E2 -1819.829} C_VEL
LIN {X 0,Y 580.169,Z 290.689,A -85,B 0,C 180,E1 -1822.057,E2 -1822.057} C_VEL
LIN {X 0,Y 580.273,Z 283.83,A -85,B 0,C 180,E1 -1825.082,E2 -1825.082} C_VEL
LIN {X 0,Y 580.254,Z 277.031,A -85,B 0,C 180,E1 -1827.85,E2 -1827.85} C_VEL
LIN {X 0,Y 580.308,Z 272.202,A -85,B 0,C 180,E1 -1829.872,E2 -1829.872} C_VEL
LIN {X 0,Y 580.296,Z 272.203,A -85,B 0,C 180,E1 -1833.025,E2 -1833.025} C_VEL
LIN {X 0,Y 580.253,Z 272.21,A -85,B 0,C 180,E1 -1835.757,E2 -1835.757} C_VEL
LIN {X 0,Y 580.292,Z 272.205,A -85,B 0,C 180,E1 -1838.147,E2 -1838.147} C_VEL
LIN {X 0,Y 580.302,Z 272.203,A -85,B 0,C 180,E1 -1840.844,E2 -1840.844} C_VEL
LIN {X 0,Y 580.284,Z 272.204,A -85,B 0,C 180,E1 -1843.658,E2 -1843.658} C_VEL
LIN {X 0,Y 580.279,Z 272.206,A -85,B 0,C 180,E1 -1846.61,E2 -1846.61} C_VEL
LIN {X 0,Y 580.303,Z 272.202,A -85,B 0,C 180,E1 -1849.157,E2 -1849.157} C_VEL
LIN {X 0,Y 580.292,Z 272.204,A -85,B 0,C 180,E1 -1851.927,E2 -1851.927} C_VEL
LIN {X 0,Y 580.253,Z 272.209,A -85,B 0,C 180,E1 -1854.453,E2 -1854.453} C_VEL
LIN {X 0,Y 580.293,Z 272.206,A -85,B 0,C 180,E1 -1856.975,E2 -1856.975} C_VEL
LIN {X 0,Y 580.3,Z 272.204,A -85,B 0,C 180,E1 -1859.425,E2 -1859.425} C_VEL
LIN {X 0,Y 580.332,Z 272.401,A -85,B 0,C 180,E1 -1861.471,E2 -1861.471} C_VEL
LIN {X 0,Y 581.227,Z 277.014,A -85,B 0,C 180,E1 -1862.34,E2 -1862.34} C_VEL
LIN {X 0,Y 581.006,Z 292.366,A -85,B 0,C 180,E1 -1864.952,E2 -1864.952} C_VEL
LIN {X 0,Y 580.805,Z 310.823,A -85,B 0,C 180,E1 -1867.969,E2 -1867.969} C_VEL
LIN {X 0,Y 580.62,Z 329.286,A -85,B 0,C 180,E1 -1870.924,E2 -1870.924} C_VEL
LIN {X 0,Y 580.487,Z 348.902,A -85,B 0,C 180,E1 -1874.012,E2 -1874.012} C_VEL
LIN {X 0,Y 580.353,Z 368.519,A -85,B 0,C 180,E1 -1877.054,E2 -1877.054} C_VEL
LIN {X 0,Y 580.326,Z 372.199,A -85,B 0,C 180,E1 -1877.598,E2 -1877.598} C_VEL
LIN {X 0,Y 580.798,Z 377.607,A -85,B 0,C 180,E1 -1877.686,E2 -1877.686} C_VEL
LIN {X 0,Y 580.762,Z 390.689,A -85,B 0,C 180,E1 -1877.973,E2 -1877.973} C_VEL
LIN {X 0,Y 580.664,Z 403.911,A -85,B 0,C 180,E1 -1878.418,E2 -1878.418} C_VEL
LIN {X 0,Y 580.576,Z 414.929,A -85,B 0,C 180,E1 -1878.92,E2 -1878.92} C_VEL
LIN {X 0,Y 580.469,Z 425.584,A -85,B 0,C 180,E1 -1879.536,E2 -1879.536} C_VEL
LIN {X 0,Y 580.38,Z 436.473,A -85,B 0,C 180,E1 -1880.327,E2 -1880.327} C_VEL
LIN {X 0,Y 580.272,Z 447.112,A -85,B 0,C 180,E1 -1881.292,E2 -1881.292} C_VEL
LIN {X 0,Y 580.222,Z 454.96,A -85,B 0,C 180,E1 -1882.168,E2 -1882.168} C_VEL
LIN {X 0,Y 580.154,Z 462.652,A -85,B 0,C 180,E1 -1883.222,E2 -1883.222} C_VEL
LIN {X 0,Y 580.139,Z 469.68,A -85,B 0,C 180,E1 -1884.438,E2 -1884.438} C_VEL
LIN {X 0,Y 580.108,Z 474.371,A -85,B 0,C 180,E1 -1885.483,E2 -1885.483} C_VEL
LIN {X 0,Y 580.123,Z 477.958,A -85,B 0,C 180,E1 -1886.527,E2 -1886.527} C_VEL
LIN {X 0,Y 580.043,Z 479.81,A -85,B 0,C 180,E1 -1887.222,E2 -1887.222} C_VEL
LIN {X 0,Y 580.04,Z 481.2,A -85,B 0,C 180,E1 -1887.917,E2 -1887.917} C_VEL
LIN {X 0,Y 580.04,Z 482.785,A -85,B 0,C 180,E1 -1889.306,E2 -1889.306} C_VEL
LIN {X 0,Y 580.037,Z 483,A -85,B 0,C 180,E1 -1890,E2 -1890} C_VEL
LIN {X 0,Y 580.047,Z 482.185,A -85,B 0,C 180,E1 -1891.389,E2 -1891.389} C_VEL
LIN {X 0,Y 580.04,Z 481.199,A -85,B 0,C 180,E1 -1892.083,E2 -1892.083} C_VEL
LIN {X 0,Y 580.043,Z 479.808,A -85,B 0,C 180,E1 -1892.778,E2 -1892.778} C_VEL
LIN {X 0,Y 580.11,Z 476.896,A -85,B 0,C 180,E1 -1893.821,E2 -1893.821} C_VEL
LIN {X 0,Y 580.053,Z 472.95,A -85,B 0,C 180,E1 -1894.865,E2 -1894.865} C_VEL
LIN {X 0,Y 580.139,Z 466.877,A -85,B 0,C 180,E1 -1896.085,E2 -1896.085} C_VEL
LIN {X 0,Y 580.185,Z 460.238,A -85,B 0,C 180,E1 -1897.132,E2 -1897.132} C_VEL
LIN {X 0,Y 580.251,Z 451.991,A -85,B 0,C 180,E1 -1898.182,E2 -1898.182} C_VEL
LIN {X 0,Y 580.308,Z 443.537,A -85,B 0,C 180,E1 -1899.058,E2 -1899.058} C_VEL
LIN {X 0,Y 580.423,Z 433.096,A -85,B 0,C 180,E1 -1899.936,E2 -1899.936} C_VEL
LIN {X 0,Y 580.529,Z 422.754,A -85,B 0,C 180,E1 -1900.639,E2 -1900.639} C_VEL
LIN {X 0,Y 580.58,Z 411.43,A -85,B 0,C 180,E1 -1901.255,E2 -1901.255} C_VEL
LIN {X 0,Y 580.657,Z 399.77,A -85,B 0,C 180,E1 -1901.741,E2 -1901.741} C_VEL
LIN {X 0,Y 580.737,Z 386.351,A -85,B 0,C 180,E1 -1902.138,E2 -1902.138} C_VEL
LIN {X 0,Y 580.615,Z 374.221,A -85,B 0,C 180,E1 -1902.368,E2 -1902.368} C_VEL
LIN {X 0,Y 580.313,Z 371.981,A -85,B 0,C 180,E1 -1902.414,E2 -1902.414} C_VEL
LIN {X 0,Y 580.424,Z 354.672,A -85,B 0,C 180,E1 -1905.09,E2 -1905.09} C_VEL
LIN {X 0,Y 580.539,Z 336.209,A -85,B 0,C 180,E1 -1907.981,E2 -1907.981} C_VEL
LIN {X 0,Y 580.707,Z 318.911,A -85,B 0,C 180,E1 -1910.73,E2 -1910.73} C_VEL
LIN {X 0,Y 580.898,Z 301.592,A -85,B 0,C 180,E1 -1913.531,E2 -1913.531} C_VEL
LIN {X 0,Y 581.106,Z 283.63,A -85,B 0,C 180,E1 -1916.495,E2 -1916.495} C_VEL
LIN {X 0,Y 581.173,Z 276.716,A -85,B 0,C 180,E1 -1917.654,E2 -1917.654} C_VEL
LIN {X 0,Y 580.294,Z 272.205,A -85,B 0,C 180,E1 -1918.531,E2 -1918.531} C_VEL
LIN {X 0,Y 580.28,Z 272.205,A -85,B 0,C 180,E1 -1921.385,E2 -1921.385} C_VEL
LIN {X 0,Y 580.285,Z 272.204,A -85,B 0,C 180,E1 -1923.857,E2 -1923.857} C_VEL
LIN {X 0,Y 580.303,Z 272.202,A -85,B 0,C 180,E1 -1926.934,E2 -1926.934} C_VEL
LIN {X 0,Y 580.298,Z 272.203,A -85,B 0,C 180,E1 -1929.933,E2 -1929.933} C_VEL
LIN {X 0,Y 580.281,Z 272.207,A -85,B 0,C 180,E1 -1932.706,E2 -1932.706} C_VEL
LIN {X 0,Y 580.276,Z 272.205,A -85,B 0,C 180,E1 -1935.609,E2 -1935.609} C_VEL
LIN {X 0,Y 580.284,Z 272.205,A -85,B 0,C 180,E1 -1938.231,E2 -1938.231} C_VEL
LIN {X 0,Y 580.29,Z 272.204,A -85,B 0,C 180,E1 -1940.965,E2 -1940.965} C_VEL
LIN {X 0,Y 580.274,Z 272.207,A -85,B 0,C 180,E1 -1943.596,E2 -1943.596} C_VEL
LIN {X 0,Y 580.305,Z 272.202,A -85,B 0,C 180,E1 -1946.144,E2 -1946.144} C_VEL
LIN {X 0,Y 580.281,Z 272.207,A -85,B 0,C 180,E1 -1948.614,E2 -1948.614} C_VEL
LIN {X 0,Y 580.209,Z 272.216,A -85,B 0,C 180,E1 -1951.019,E2 -1951.019} C_VEL
LIN {X 0,Y 580.125,Z 272.513,A -85,B 0,C 180,E1 -1951.311,E2 -1951.311} C_VEL
LIN {X 0,Y 580.13,Z 279.247,A -85,B 0,C 180,E1 -1953.699,E2 -1953.699} C_VEL
LIN {X 0,Y 580.151,Z 286.597,A -85,B 0,C 180,E1 -1956.436,E2 -1956.436} C_VEL
LIN {X 0,Y 580.136,Z 293.934,A -85,B 0,C 180,E1 -1959.431,E2 -1959.431} C_VEL
LIN {X 0,Y 580.127,Z 301.15,A -85,B 0,C 180,E1 -1962.369,E2 -1962.369} C_VEL
LIN {X 0,Y 580.105,Z 308.366,A -85,B 0,C 180,E1 -1965.26,E2 -1965.26} C_VEL
LIN {X 0,Y 580.085,Z 315.582,A -85,B 0,C 180,E1 -1968.113,E2 -1968.113} C_VEL
LIN {X 0,Y 580.031,Z 322.799,A -85,B 0,C 180,E1 -1970.936,E2 -1970.936} C_VEL
LIN {X 0,Y 580.068,Z 327.729,A -85,B 0,C 180,E1 -1972.843,E2 -1972.843} C_VEL
LIN {X 0,Y 580.305,Z 335.774,A -85,B 0,C 180,E1 -1973.119,E2 -1973.119} C_VEL
LIN {X 0,Y 580.253,Z 344.826,A -85,B 0,C 180,E1 -1973.553,E2 -1973.553} C_VEL
LIN {X 0,Y 580.206,Z 353.02,A -85,B 0,C 180,E1 -1974.09,E2 -1974.09} C_VEL
LIN {X 0,Y 580.165,Z 361.066,A -85,B 0,C 180,E1 -1974.786,E2 -1974.786} C_VEL
LIN {X 0,Y 580.151,Z 367.22,A -85,B 0,C 180,E1 -1975.483,E2 -1975.483} C_VEL
LIN {X 0,Y 580.157,Z 372.065,A -85,B 0,C 180,E1 -1976.179,E2 -1976.179} C_VEL
LIN {X 0,Y 580.095,Z 375.834,A -85,B 0,C 180,E1 -1976.874,E2 -1976.874} C_VEL
LIN {X 0,Y 580.049,Z 379.827,A -85,B 0,C 180,E1 -1977.916,E2 -1977.916} C_VEL
LIN {X 0,Y 580.047,Z 381.568,A -85,B 0,C 180,E1 -1978.611,E2 -1978.611} C_VEL
LIN {X 0,Y 580.041,Z 382.616,A -85,B 0,C 180,E1 -1979.305,E2 -1979.305} C_VEL
LIN {X 0,Y 580.038,Z 382.996,A -85,B 0,C 180,E1 -1979.999,E2 -1979.999} C_VEL
LIN {X 0,Y 580.04,Z 382.713,A -85,B 0,C 180,E1 -1980.693,E2 -1980.693} C_VEL
LIN {X 0,Y 580.048,Z 381.764,A -85,B 0,C 180,E1 -1981.388,E2 -1981.388} C_VEL
LIN {X 0,Y 580.092,Z 378.997,A -85,B 0,C 180,E1 -1982.429,E2 -1982.429} C_VEL
LIN {X 0,Y 580.095,Z 376.239,A -85,B 0,C 180,E1 -1983.124,E2 -1983.124} C_VEL
LIN {X 0,Y 580.133,Z 371.536,A -85,B 0,C 180,E1 -1983.993,E2 -1983.993} C_VEL
LIN {X 0,Y 580.171,Z 365.146,A -85,B 0,C 180,E1 -1984.863,E2 -1984.863} C_VEL
LIN {X 0,Y 580.138,Z 358.358,A -85,B 0,C 180,E1 -1985.561,E2 -1985.561} C_VEL
LIN {X 0,Y 580.241,Z 350.674,A -85,B 0,C 180,E1 -1986.17,E2 -1986.17} C_VEL
LIN {X 0,Y 580.266,Z 341.688,A -85,B 0,C 180,E1 -1986.704,E2 -1986.704} C_VEL
LIN {X 0,Y 580.316,Z 332.719,A -85,B 0,C 180,E1 -1987.086,E2 -1987.086} C_VEL
LIN {X 0,Y 580.055,Z 327.659,A -85,B 0,C 180,E1 -1987.264,E2 -1987.264} C_VEL
LIN {X 0,Y 580.061,Z 321.23,A -85,B 0,C 180,E1 -1989.765,E2 -1989.765} C_VEL
LIN {X 0,Y 580.084,Z 315.816,A -85,B 0,C 180,E1 -1991.885,E2 -1991.885} C_VEL
LIN {X 0,Y 580.117,Z 308.597,A -85,B 0,C 180,E1 -1994.738,E2 -1994.738} C_VEL
LIN {X 0,Y 580.12,Z 301.062,A -85,B 0,C 180,E1 -1997.756,E2 -1997.756} C_VEL
LIN {X 0,Y 580.145,Z 294.158,A -85,B 0,C 180,E1 -2000.566,E2 -2000.566} C_VEL
LIN {X 0,Y 580.142,Z 293.842,A -85,B 0,C 180,E1 -2000.697,E2 -2000.697} C_VEL
LIN {X 0,Y 579.471,Z 292.576,A -85,B 0,C 180,E1 -2001.261,E2 -2001.261} C_VEL
LIN {X 0,Y 576.604,Z 290.722,A -85,B 0,C 180,E1 -2002.182,E2 -2002.182} C_VEL
LIN {X 0,Y 574.188,Z 289.139,A -85,B 0,C 180,E1 -2002.923,E2 -2002.923} C_VEL
LIN {X 0,Y 573.163,Z 287.812,A -85,B 0,C 180,E1 -2003.493,E2 -2003.493} C_VEL
LIN {X 0,Y 573.086,Z 287.341,A -85,B 0,C 180,E1 -2003.685,E2 -2003.685} C_VEL
LIN {X 0,Y 573.146,Z 281.292,A -85,B 0,C 180,E1 -2006.194,E2 -2006.194} C_VEL
LIN {X 0,Y 573.177,Z 274.322,A -85,B 0,C 180,E1 -2008.967,E2 -2008.967} C_VEL
LIN {X 0,Y 573.197,Z 273.089,A -85,B 0,C 180,E1 -2009.479,E2 -2009.479} C_VEL
LIN {X 0,Y 573.237,Z 273.076,A -85,B 0,C 180,E1 -2012.645,E2 -2012.645} C_VEL
LIN {X 0,Y 573.18,Z 273.091,A -85,B 0,C 180,E1 -2015.188,E2 -2015.188} C_VEL
LIN {X 0,Y 573.22,Z 273.078,A -85,B 0,C 180,E1 -2017.807,E2 -2017.807} C_VEL
LIN {X 0,Y 573.238,Z 273.08,A -85,B 0,C 180,E1 -2020.524,E2 -2020.524} C_VEL
LIN {X 0,Y 573.202,Z 273.081,A -85,B 0,C 180,E1 -2023.361,E2 -2023.361} C_VEL
LIN {X 0,Y 573.231,Z 273.083,A -85,B 0,C 180,E1 -2026.331,E2 -2026.331} C_VEL
LIN {X 0,Y 573.266,Z 273.072,A -85,B 0,C 180,E1 -2029.476,E2 -2029.476} C_VEL
LIN {X 0,Y 573.229,Z 273.085,A -85,B 0,C 180,E1 -2032.192,E2 -2032.192} C_VEL
LIN {X 0,Y 573.259,Z 273.073,A -85,B 0,C 180,E1 -2034.816,E2 -2034.816} C_VEL
LIN {X 0,Y 573.248,Z 273.077,A -85,B 0,C 180,E1 -2037.354,E2 -2037.354} C_VEL
LIN {X 0,Y 573.248,Z 273.082,A -85,B 0,C 180,E1 -2039.824,E2 -2039.824} C_VEL
LIN {X 0,Y 573.28,Z 273.072,A -85,B 0,C 180,E1 -2042.234,E2 -2042.234} C_VEL
LIN {X 0,Y 573.258,Z 273.078,A -85,B 0,C 180,E1 -2045.121,E2 -2045.121} C_VEL
LIN {X 0,Y 573.229,Z 273.08,A -85,B 0,C 180,E1 -2047.662,E2 -2047.662} C_VEL
LIN {X 0,Y 573.245,Z 273.075,A -85,B 0,C 180,E1 -2049.923,E2 -2049.923} C_VEL
LIN {X 0,Y 573.249,Z 273.082,A -85,B 0,C 180,E1 -2052.989,E2 -2052.989} C_VEL
LIN {X 0,Y 573.262,Z 273.073,A -85,B 0,C 180,E1 -2055.807,E2 -2055.807} C_VEL
LIN {X 0,Y 573.25,Z 273.081,A -85,B 0,C 180,E1 -2058.745,E2 -2058.745} C_VEL
LIN {X 0,Y 573.265,Z 273.072,A -85,B 0,C 180,E1 -2061.54,E2 -2061.54} C_VEL
LIN {X 0,Y 573.274,Z 273.079,A -85,B 0,C 180,E1 -2064.372,E2 -2064.372} C_VEL
LIN {X 0,Y 573.301,Z 273.073,A -85,B 0,C 180,E1 -2067.892,E2 -2067.892} C_VEL
LIN {X 0,Y 573.305,Z 273.076,A -85,B 0,C 180,E1 -2070,E2 -2070} C_VEL
LIN {X 0,Y 573.264,Z 273.072,A -85,B 0,C 180,E1 -2072.811,E2 -2072.811} C_VEL
LIN {X 0,Y 573.276,Z 273.079,A -85,B 0,C 180,E1 -2075.628,E2 -2075.628} C_VEL
LIN {X 0,Y 573.266,Z 273.072,A -85,B 0,C 180,E1 -2078.46,E2 -2078.46} C_VEL
LIN {X 0,Y 573.259,Z 273.081,A -85,B 0,C 180,E1 -2081.312,E2 -2081.312} C_VEL
LIN {X 0,Y 573.27,Z 273.072,A -85,B 0,C 180,E1 -2084.425,E2 -2084.425} C_VEL
LIN {X 0,Y 573.248,Z 273.082,A -85,B 0,C 180,E1 -2087.112,E2 -2087.112} C_VEL
LIN {X 0,Y 573.245,Z 273.075,A -85,B 0,C 180,E1 -2090.077,E2 -2090.077} C_VEL
LIN {X 0,Y 573.229,Z 273.081,A -85,B 0,C 180,E1 -2092.338,E2 -2092.338} C_VEL
LIN {X 0,Y 573.247,Z 273.075,A -85,B 0,C 180,E1 -2095.411,E2 -2095.411} C_VEL
LIN {X 0,Y 573.255,Z 273.078,A -85,B 0,C 180,E1 -2098.033,E2 -2098.033} C_VEL
LIN {X 0,Y 573.235,Z 273.077,A -85,B 0,C 180,E1 -2100.886,E2 -2100.886} C_VEL
LIN {X 0,Y 573.279,Z 273.073,A -85,B 0,C 180,E1 -2103.529,E2 -2103.529} C_VEL
LIN {X 0,Y 573.252,Z 273.081,A -85,B 0,C 180,E1 -2106.049,E2 -2106.049} C_VEL
LIN {X 0,Y 573.242,Z 273.075,A -85,B 0,C 180,E1 -2108.702,E2 -2108.702} C_VEL
LIN {X 0,Y 573.222,Z 273.085,A -85,B 0,C 180,E1 -2111.458,E2 -2111.458} C_VEL
LIN {X 0,Y 573.217,Z 273.078,A -85,B 0,C 180,E1 -2114.336,E2 -2114.336} C_VEL
LIN {X 0,Y 573.229,Z 273.084,A -85,B 0,C 180,E1 -2117.36,E2 -2117.36} C_VEL
LIN {X 0,Y 573.225,Z 273.078,A -85,B 0,C 180,E1 -2120.393,E2 -2120.393} C_VEL
LIN {X 0,Y 573.225,Z 273.084,A -85,B 0,C 180,E1 -2123.077,E2 -2123.077} C_VEL
LIN {X 0,Y 573.236,Z 273.075,A -85,B 0,C 180,E1 -2125.671,E2 -2125.671} C_VEL
LIN {X 0,Y 573.219,Z 273.08,A -85,B 0,C 180,E1 -2128.185,E2 -2128.185} C_VEL
LIN {X 0,Y 573.271,Z 273.099,A -85,B 0,C 180,E1 -2130.2,E2 -2130.2} C_VEL
LIN {X 0,Y 573.178,Z 279.655,A -85,B 0,C 180,E1 -2133.022,E2 -2133.022} C_VEL
LIN {X 0,Y 573.177,Z 285.218,A -85,B 0,C 180,E1 -2135.363,E2 -2135.363} C_VEL
LIN {X 0,Y 573.1,Z 290.484,A -85,B 0,C 180,E1 -2137.658,E2 -2137.658} C_VEL
LIN {X 0,Y 573.043,Z 295.747,A -85,B 0,C 180,E1 -2139.917,E2 -2139.917} C_VEL
LIN {X 0,Y 573.022,Z 302.96,A -85,B 0,C 180,E1 -2142.882,E2 -2142.882} C_VEL
LIN {X 0,Y 573.045,Z 310.176,A -85,B 0,C 180,E1 -2145.802,E2 -2145.802} C_VEL
LIN {X 0,Y 573.013,Z 317.87,A -85,B 0,C 180,E1 -2148.873,E2 -2148.873} C_VEL
LIN {X 0,Y 572.985,Z 324.609,A -85,B 0,C 180,E1 -2151.537,E2 -2151.537} C_VEL
LIN {X 0,Y 572.963,Z 327.78,A -85,B 0,C 180,E1 -2152.756,E2 -2152.756} C_VEL
LIN {X 0,Y 573.269,Z 335.892,A -85,B 0,C 180,E1 -2153.038,E2 -2153.038} C_VEL
LIN {X 0,Y 573.183,Z 344.747,A -85,B 0,C 180,E1 -2153.473,E2 -2153.473} C_VEL
LIN {X 0,Y 573.175,Z 351.834,A -85,B 0,C 180,E1 -2153.93,E2 -2153.93} C_VEL
LIN {X 0,Y 573.036,Z 359.254,A -85,B 0,C 180,E1 -2154.547,E2 -2154.547} C_VEL
LIN {X 0,Y 573.082,Z 364.34,A -85,B 0,C 180,E1 -2155.076,E2 -2155.076} C_VEL
LIN {X 0,Y 573.037,Z 369.767,A -85,B 0,C 180,E1 -2155.781,E2 -2155.781} C_VEL
LIN {X 0,Y 573.062,Z 374.057,A -85,B 0,C 180,E1 -2156.485,E2 -2156.485} C_VEL
LIN {X 0,Y 572.972,Z 377.379,A -85,B 0,C 180,E1 -2157.189,E2 -2157.189} C_VEL
LIN {X 0,Y 572.952,Z 379.857,A -85,B 0,C 180,E1 -2157.892,E2 -2157.892} C_VEL
LIN {X 0,Y 572.947,Z 381.571,A -85,B 0,C 180,E1 -2158.595,E2 -2158.595} C_VEL
LIN {X 0,Y 572.941,Z 382.585,A -85,B 0,C 180,E1 -2159.298,E2 -2159.298} C_VEL
LIN {X 0,Y 572.939,Z 382.954,A -85,B 0,C 180,E1 -2160.001,E2 -2160.001} C_VEL
LIN {X 0,Y 572.941,Z 382.687,A -85,B 0,C 180,E1 -2160.704,E2 -2160.704} C_VEL
LIN {X 0,Y 572.948,Z 381.76,A -85,B 0,C 180,E1 -2161.407,E2 -2161.407} C_VEL
LIN {X 0,Y 573.016,Z 378.996,A -85,B 0,C 180,E1 -2162.461,E2 -2162.461} C_VEL
LIN {X 0,Y 573.013,Z 376.243,A -85,B 0,C 180,E1 -2163.165,E2 -2163.165} C_VEL
LIN {X 0,Y 573.037,Z 371.5,A -85,B 0,C 180,E1 -2164.045,E2 -2164.045} C_VEL
LIN {X 0,Y 573.112,Z 366.529,A -85,B 0,C 180,E1 -2164.749,E2 -2164.749} C_VEL
